LIN {X 0,Y 684.973,Z 1061.828,A -85,B 0,C 180,E1 30898.463,E2 30898.463} C_VEL
LIN {X 0,Y 683.766,Z 1083.483,A -85,B 0,C 180,E1 30896.498,E2 30896.498} C_VEL
LIN {X 0,Y 682.983,Z 1099.696,A -85,B 0,C 180,E1 30894.844,E2 30894.844} C_VEL
LIN {X 0,Y 682.192,Z 1116.492,A -85,B 0,C 180,E1 30892.946,E2 30892.946} C_VEL
LIN {X 0,Y 681.497,Z 1132.898,A -85,B 0,C 180,E1 30890.835,E2 30890.835} C_VEL
LIN {X 0,Y 681.037,Z 1145.572,A -85,B 0,C 180,E1 30889,E2 30889} C_VEL
LIN {X 0,Y 680.644,Z 1157.898,A -85,B 0,C 180,E1 30886.992,E2 30886.992} C_VEL
LIN {X 0,Y 680.337,Z 1169.84,A -85,B 0,C 180,E1 30884.729,E2 30884.729} C_VEL
LIN {X 0,Y 680.158,Z 1178.438,A -85,B 0,C 180,E1 30882.825,E2 30882.825} C_VEL
LIN {X 0,Y 680.019,Z 1186.223,A -85,B 0,C 180,E1 30880.819,E2 30880.819} C_VEL
LIN {X 0,Y 679.964,Z 1193.354,A -85,B 0,C 180,E1 30878.541,E2 30878.541} C_VEL
LIN {X 0,Y 679.926,Z 1198.83,A -85,B 0,C 180,E1 30876.216,E2 30876.216} C_VEL
LIN {X 0,Y 679.913,Z 1202.374,A -85,B 0,C 180,E1 30874.048,E2 30874.048} C_VEL
LIN {X 0,Y 679.907,Z 1204.494,A -85,B 0,C 180,E1 30871.77,E2 30871.77} C_VEL
LIN {X 0,Y 679.891,Z 1204.872,A -85,B 0,C 180,E1 30869.494,E2 30869.494} C_VEL
LIN {X 0,Y 679.907,Z 1203.956,A -85,B 0,C 180,E1 30867.471,E2 30867.471} C_VEL
LIN {X 0,Y 679.911,Z 1201.428,A -85,B 0,C 180,E1 30865.276,E2 30865.276} C_VEL
LIN {X 0,Y 679.934,Z 1197.152,A -85,B 0,C 180,E1 30862.989,E2 30862.989} C_VEL
LIN {X 0,Y 679.978,Z 1191.385,A -85,B 0,C 180,E1 30860.777,E2 30860.777} C_VEL
LIN {X 0,Y 680.067,Z 1184.278,A -85,B 0,C 180,E1 30858.638,E2 30858.638} C_VEL
LIN {X 0,Y 680.24,Z 1173.938,A -85,B 0,C 180,E1 30856.138,E2 30856.138} C_VEL
LIN {X 0,Y 680.464,Z 1164.538,A -85,B 0,C 180,E1 30854.227,E2 30854.227} C_VEL
LIN {X 0,Y 680.75,Z 1154.23,A -85,B 0,C 180,E1 30852.388,E2 30852.388} C_VEL
LIN {X 0,Y 681.149,Z 1141.939,A -85,B 0,C 180,E1 30850.447,E2 30850.447} C_VEL
LIN {X 0,Y 681.795,Z 1125.467,A -85,B 0,C 180,E1 30848.177,E2 30848.177} C_VEL
LIN {X 0,Y 682.441,Z 1111.072,A -85,B 0,C 180,E1 30846.423,E2 30846.423} C_VEL
LIN {X 0,Y 683.272,Z 1093.721,A -85,B 0,C 180,E1 30844.518,E2 30844.518} C_VEL
LIN {X 0,Y 684.268,Z 1074.724,A -85,B 0,C 180,E1 30842.679,E2 30842.679} C_VEL
LIN {X 0,Y 685.156,Z 1057.953,A -85,B 0,C 180,E1 30841.212,E2 30841.212} C_VEL
LIN {X 0,Y 686.26,Z 1038.594,A -85,B 0,C 180,E1 30839.679,E2 30839.679} C_VEL
LIN {X 0,Y 687.621,Z 1015.181,A -85,B 0,C 180,E1 30838.043,E2 30838.043} C_VEL
LIN {X 0,Y 688.735,Z 995.45,A -85,B 0,C 180,E1 30836.818,E2 30836.818} C_VEL
LIN {X 0,Y 689.843,Z 975.498,A -85,B 0,C 180,E1 30835.709,E2 30835.709} C_VEL
LIN {X 0,Y 691.118,Z 951.696,A -85,B 0,C 180,E1 30834.54,E2 30834.54} C_VEL
LIN {X 0,Y 692.334,Z 926.433,A -85,B 0,C 180,E1 30833.487,E2 30833.487} C_VEL
LIN {X 0,Y 693.317,Z 904.148,A -85,B 0,C 180,E1 30832.695,E2 30832.695} C_VEL
LIN {X 0,Y 694.253,Z 881.072,A -85,B 0,C 180,E1 30832.002,E2 30832.002} C_VEL
LIN {X 0,Y 695.165,Z 854.15,A -85,B 0,C 180,E1 30831.357,E2 30831.357} C_VEL
LIN {X 0,Y 695.824,Z 826.984,A -85,B 0,C 180,E1 30830.881,E2 30830.881} C_VEL
LIN {X 0,Y 698.219,Z 604.951,A -85,B 0,C 180,E1 30828.078,E2 30828.078} C_VEL
LIN {X 0,Y 700.483,Z 400.768,A -85,B 0,C 180,E1 30825.432,E2 30825.432} C_VEL
LIN {X 0,Y 700.65,Z 371.916,A -85,B 0,C 180,E1 30825.038,E2 30825.038} C_VEL
LIN {X 0,Y 697.923,Z 362.231,A -85,B 0,C 180,E1 30824.675,E2 30824.675} C_VEL
LIN {X 0,Y 690.097,Z 350.376,A -85,B 0,C 180,E1 30823.819,E2 30823.819} C_VEL
LIN {X 0,Y 683.625,Z 336.783,A -85,B 0,C 180,E1 30822.171,E2 30822.171} C_VEL
LIN {X 0,Y 681.952,Z 333.226,A -85,B 0,C 180,E1 30821.731,E2 30821.731} C_VEL
LIN {X 0,Y 680.493,Z 329.763,A -85,B 0,C 180,E1 30821.314,E2 30821.314} C_VEL
LIN {X 0,Y 680.459,Z 329.472,A -85,B 0,C 180,E1 30821.171,E2 30821.171} C_VEL
LIN {X 0,Y 680.503,Z 329.468,A -85,B 0,C 180,E1 30818.107,E2 30818.107} C_VEL
LIN {X 0,Y 680.45,Z 329.469,A -85,B 0,C 180,E1 30815.361,E2 30815.361} C_VEL
LIN {X 0,Y 680.488,Z 329.464,A -85,B 0,C 180,E1 30812.657,E2 30812.657} C_VEL
LIN {X 0,Y 680.469,Z 329.468,A -85,B 0,C 180,E1 30809.557,E2 30809.557} C_VEL
LIN {X 0,Y 680.449,Z 329.447,A -85,B 0,C 180,E1 30807.005,E2 30807.005} C_VEL
LIN {X 0,Y 680.526,Z 329.463,A -85,B 0,C 180,E1 30804.108,E2 30804.108} C_VEL
LIN {X 0,Y 680.462,Z 329.465,A -85,B 0,C 180,E1 30801.191,E2 30801.191} C_VEL
LIN {X 0,Y 680.459,Z 329.459,A -85,B 0,C 180,E1 30798.595,E2 30798.595} C_VEL
LIN {X 0,Y 680.526,Z 329.458,A -85,B 0,C 180,E1 30795.598,E2 30795.598} C_VEL
LIN {X 0,Y 680.454,Z 329.448,A -85,B 0,C 180,E1 30792.734,E2 30792.734} C_VEL
LIN {X 0,Y 680.494,Z 329.459,A -85,B 0,C 180,E1 30789.985,E2 30789.985} C_VEL
LIN {X 0,Y 680.474,Z 329.447,A -85,B 0,C 180,E1 30786.92,E2 30786.92} C_VEL
LIN {X 0,Y 680.458,Z 329.464,A -85,B 0,C 180,E1 30784.298,E2 30784.298} C_VEL
LIN {X 0,Y 680.527,Z 329.443,A -85,B 0,C 180,E1 30781.347,E2 30781.347} C_VEL
LIN {X 0,Y 680.461,Z 329.465,A -85,B 0,C 180,E1 30778.4,E2 30778.4} C_VEL
LIN {X 0,Y 680.49,Z 329.442,A -85,B 0,C 180,E1 30775.618,E2 30775.618} C_VEL
LIN {X 0,Y 680.477,Z 329.463,A -85,B 0,C 180,E1 30772.485,E2 30772.485} C_VEL
LIN {X 0,Y 680.465,Z 329.451,A -85,B 0,C 180,E1 30769.758,E2 30769.758} C_VEL
LIN {X 0,Y 680.527,Z 329.454,A -85,B 0,C 180,E1 30766.749,E2 30766.749} C_VEL
LIN {X 0,Y 680.462,Z 329.464,A -85,B 0,C 180,E1 30763.876,E2 30763.876} C_VEL
LIN {X 0,Y 680.512,Z 329.449,A -85,B 0,C 180,E1 30761.051,E2 30761.051} C_VEL
LIN {X 0,Y 680.475,Z 329.464,A -85,B 0,C 180,E1 30757.994,E2 30757.994} C_VEL
LIN {X 0,Y 680.474,Z 329.458,A -85,B 0,C 180,E1 30755.238,E2 30755.238} C_VEL
LIN {X 0,Y 680.512,Z 329.467,A -85,B 0,C 180,E1 30752.144,E2 30752.144} C_VEL
LIN {X 0,Y 680.466,Z 329.463,A -85,B 0,C 180,E1 30749.39,E2 30749.39} C_VEL
LIN {X 0,Y 679.48,Z 329.589,A -85,B 0,C 180,E1 30748.742,E2 30748.742} C_VEL
LIN {X 0,Y 673.099,Z 330.39,A -85,B 0,C 180,E1 30746.924,E2 30746.924} C_VEL
LIN {X 0,Y 672.588,Z 330.454,A -85,B 0,C 180,E1 30746.452,E2 30746.452} C_VEL
LIN {X 0,Y 672.558,Z 330.625,A -85,B 0,C 180,E1 30745.555,E2 30745.555} C_VEL
LIN {X 0,Y 673.93,Z 334.074,A -85,B 0,C 180,E1 30745.129,E2 30745.129} C_VEL
LIN {X 0,Y 677.255,Z 341.083,A -85,B 0,C 180,E1 30744.248,E2 30744.248} C_VEL
LIN {X 0,Y 689.877,Z 359.457,A -85,B 0,C 180,E1 30742.854,E2 30742.854} C_VEL
LIN {X 0,Y 695.097,Z 367.633,A -85,B 0,C 180,E1 30742.294,E2 30742.294} C_VEL
LIN {X 0,Y 692.503,Z 574.54,A -85,B 0,C 180,E1 30739.585,E2 30739.585} C_VEL
LIN {X 0,Y 689.933,Z 798.204,A -85,B 0,C 180,E1 30736.745,E2 30736.745} C_VEL
LIN {X 0,Y 689.322,Z 828.688,A -85,B 0,C 180,E1 30736.308,E2 30736.308} C_VEL
LIN {X 0,Y 688.525,Z 853.699,A -85,B 0,C 180,E1 30735.805,E2 30735.805} C_VEL
LIN {X 0,Y 687.518,Z 880.23,A -85,B 0,C 180,E1 30735.112,E2 30735.112} C_VEL
LIN {X 0,Y 686.268,Z 907.112,A -85,B 0,C 180,E1 30734.225,E2 30734.225} C_VEL
LIN {X 0,Y 685.119,Z 929.491,A -85,B 0,C 180,E1 30733.348,E2 30733.348} C_VEL
LIN {X 0,Y 683.72,Z 954.189,A -85,B 0,C 180,E1 30732.219,E2 30732.219} C_VEL
LIN {X 0,Y 682.144,Z 979.486,A -85,B 0,C 180,E1 30730.873,E2 30730.873} C_VEL
LIN {X 0,Y 680.693,Z 1002.914,A -85,B 0,C 180,E1 30729.436,E2 30729.436} C_VEL
LIN {X 0,Y 679.296,Z 1024.873,A -85,B 0,C 180,E1 30727.911,E2 30727.911} C_VEL
LIN {X 0,Y 677.913,Z 1046.47,A -85,B 0,C 180,E1 30726.215,E2 30726.215} C_VEL
LIN {X 0,Y 676.678,Z 1067.352,A -85,B 0,C 180,E1 30724.363,E2 30724.363} C_VEL
LIN {X 0,Y 675.512,Z 1086.947,A -85,B 0,C 180,E1 30722.399,E2 30722.399} C_VEL
LIN {X 0,Y 674.581,Z 1105,A -85,B 0,C 180,E1 30720.36,E2 30720.36} C_VEL
LIN {X 0,Y 673.743,Z 1122.087,A -85,B 0,C 180,E1 30718.159,E2 30718.159} C_VEL
LIN {X 0,Y 673.134,Z 1136.715,A -85,B 0,C 180,E1 30716.014,E2 30716.014} C_VEL
LIN {X 0,Y 672.647,Z 1150.472,A -85,B 0,C 180,E1 30713.696,E2 30713.696} C_VEL
LIN {X 0,Y 672.343,Z 1161.747,A -85,B 0,C 180,E1 30711.459,E2 30711.459} C_VEL
LIN {X 0,Y 672.134,Z 1170.61,A -85,B 0,C 180,E1 30709.41,E2 30709.41} C_VEL
LIN {X 0,Y 672.014,Z 1178.571,A -85,B 0,C 180,E1 30707.208,E2 30707.208} C_VEL
LIN {X 0,Y 671.96,Z 1185.341,A -85,B 0,C 180,E1 30704.829,E2 30704.829} C_VEL
LIN {X 0,Y 671.927,Z 1190.109,A -85,B 0,C 180,E1 30702.548,E2 30702.548} C_VEL
LIN {X 0,Y 671.919,Z 1193.274,A -85,B 0,C 180,E1 30700.286,E2 30700.286} C_VEL
LIN {X 0,Y 671.908,Z 1194.7,A -85,B 0,C 180,E1 30698.127,E2 30698.127} C_VEL
LIN {X 0,Y 671.913,Z 1194.819,A -85,B 0,C 180,E1 30696.236,E2 30696.236} C_VEL
LIN {X 0,Y 671.913,Z 1193.788,A -85,B 0,C 180,E1 30694.181,E2 30694.181} C_VEL
LIN {X 0,Y 671.92,Z 1190.996,A -85,B 0,C 180,E1 30691.876,E2 30691.876} C_VEL
LIN {X 0,Y 671.938,Z 1186.49,A -85,B 0,C 180,E1 30689.574,E2 30689.574} C_VEL
LIN {X 0,Y 671.998,Z 1180.619,A -85,B 0,C 180,E1 30687.356,E2 30687.356} C_VEL
LIN {X 0,Y 672.108,Z 1172.449,A -85,B 0,C 180,E1 30684.965,E2 30684.965} C_VEL
LIN {X 0,Y 672.308,Z 1163.087,A -85,B 0,C 180,E1 30682.738,E2 30682.738} C_VEL
LIN {X 0,Y 672.574,Z 1152.894,A -85,B 0,C 180,E1 30680.675,E2 30680.675} C_VEL
LIN {X 0,Y 672.996,Z 1140.618,A -85,B 0,C 180,E1 30678.517,E2 30678.517} C_VEL
LIN {X 0,Y 673.553,Z 1126.357,A -85,B 0,C 180,E1 30676.348,E2 30676.348} C_VEL
LIN {X 0,Y 674.262,Z 1110.628,A -85,B 0,C 180,E1 30674.245,E2 30674.245} C_VEL
LIN {X 0,Y 675.225,Z 1092.867,A -85,B 0,C 180,E1 30672.15,E2 30672.15} C_VEL
LIN {X 0,Y 676.3,Z 1073.164,A -85,B 0,C 180,E1 30670.104,E2 30670.104} C_VEL
LIN {X 0,Y 677.596,Z 1051.897,A -85,B 0,C 180,E1 30668.154,E2 30668.154} C_VEL
LIN {X 0,Y 678.995,Z 1029.504,A -85,B 0,C 180,E1 30666.343,E2 30666.343} C_VEL
LIN {X 0,Y 680.508,Z 1006.177,A -85,B 0,C 180,E1 30664.687,E2 30664.687} C_VEL
LIN {X 0,Y 682.022,Z 981.614,A -85,B 0,C 180,E1 30663.158,E2 30663.158} C_VEL
LIN {X 0,Y 683.636,Z 955.647,A -85,B 0,C 180,E1 30661.762,E2 30661.762} C_VEL
LIN {X 0,Y 685.083,Z 930.161,A -85,B 0,C 180,E1 30660.591,E2 30660.591} C_VEL
LIN {X 0,Y 686.276,Z 906.976,A -85,B 0,C 180,E1 30659.68,E2 30659.68} C_VEL
LIN {X 0,Y 687.523,Z 880.087,A -85,B 0,C 180,E1 30658.793,E2 30658.793} C_VEL
LIN {X 0,Y 688.539,Z 853.473,A -85,B 0,C 180,E1 30658.101,E2 30658.101} C_VEL
LIN {X 0,Y 689.323,Z 828.529,A -85,B 0,C 180,E1 30657.598,E2 30657.598} C_VEL
LIN {X 0,Y 689.945,Z 796.974,A -85,B 0,C 180,E1 30657.15,E2 30657.15} C_VEL
LIN {X 0,Y 692.503,Z 574.702,A -85,B 0,C 180,E1 30654.328,E2 30654.328} C_VEL
LIN {X 0,Y 695.099,Z 367.462,A -85,B 0,C 180,E1 30651.614,E2 30651.614} C_VEL
LIN {X 0,Y 684.64,Z 351.816,A -85,B 0,C 180,E1 30650.488,E2 30650.488} C_VEL
LIN {X 0,Y 677.093,Z 340.807,A -85,B 0,C 180,E1 30649.641,E2 30649.641} C_VEL
LIN {X 0,Y 673.916,Z 334.126,A -85,B 0,C 180,E1 30648.785,E2 30648.785} C_VEL
LIN {X 0,Y 672.529,Z 330.601,A -85,B 0,C 180,E1 30648.352,E2 30648.352} C_VEL
LIN {X 0,Y 672.5,Z 330.462,A -85,B 0,C 180,E1 30645.192,E2 30645.192} C_VEL
LIN {X 0,Y 672.483,Z 330.449,A -85,B 0,C 180,E1 30642.689,E2 30642.689} C_VEL
LIN {X 0,Y 672.525,Z 330.46,A -85,B 0,C 180,E1 30640.034,E2 30640.034} C_VEL
LIN {X 0,Y 672.507,Z 330.456,A -85,B 0,C 180,E1 30637.024,E2 30637.024} C_VEL
LIN {X 0,Y 672.486,Z 330.453,A -85,B 0,C 180,E1 30634.506,E2 30634.506} C_VEL
LIN {X 0,Y 672.522,Z 330.454,A -85,B 0,C 180,E1 30631.858,E2 30631.858} C_VEL
LIN {X 0,Y 672.507,Z 330.439,A -85,B 0,C 180,E1 30628.798,E2 30628.798} C_VEL
LIN {X 0,Y 672.49,Z 330.45,A -85,B 0,C 180,E1 30626.206,E2 30626.206} C_VEL
LIN {X 0,Y 672.56,Z 330.445,A -85,B 0,C 180,E1 30623.388,E2 30623.388} C_VEL
LIN {X 0,Y 672.5,Z 330.447,A -85,B 0,C 180,E1 30620.451,E2 30620.451} C_VEL
LIN {X 0,Y 672.493,Z 330.457,A -85,B 0,C 180,E1 30617.91,E2 30617.91} C_VEL
LIN {X 0,Y 672.587,Z 330.454,A -85,B 0,C 180,E1 30614.992,E2 30614.992} C_VEL
LIN {X 0,Y 672.495,Z 330.456,A -85,B 0,C 180,E1 30612.102,E2 30612.102} C_VEL
LIN {X 0,Y 672.499,Z 330.451,A -85,B 0,C 180,E1 30609.586,E2 30609.586} C_VEL
LIN {X 0,Y 672.576,Z 330.446,A -85,B 0,C 180,E1 30606.659,E2 30606.659} C_VEL
LIN {X 0,Y 672.496,Z 330.455,A -85,B 0,C 180,E1 30603.836,E2 30603.836} C_VEL
LIN {X 0,Y 672.507,Z 330.455,A -85,B 0,C 180,E1 30601.278,E2 30601.278} C_VEL
LIN {X 0,Y 672.544,Z 330.454,A -85,B 0,C 180,E1 30598.211,E2 30598.211} C_VEL
LIN {X 0,Y 672.495,Z 330.449,A -85,B 0,C 180,E1 30595.48,E2 30595.48} C_VEL
LIN {X 0,Y 672.532,Z 330.457,A -85,B 0,C 180,E1 30592.826,E2 30592.826} C_VEL
LIN {X 0,Y 672.516,Z 330.453,A -85,B 0,C 180,E1 30589.723,E2 30589.723} C_VEL
LIN {X 0,Y 672.497,Z 330.431,A -85,B 0,C 180,E1 30587.113,E2 30587.113} C_VEL
LIN {X 0,Y 672.589,Z 330.454,A -85,B 0,C 180,E1 30584.213,E2 30584.213} C_VEL
LIN {X 0,Y 672.501,Z 330.433,A -85,B 0,C 180,E1 30581.267,E2 30581.267} C_VEL
LIN {X 0,Y 672.509,Z 330.453,A -85,B 0,C 180,E1 30578.729,E2 30578.729} C_VEL
LIN {X 0,Y 672.572,Z 330.426,A -85,B 0,C 180,E1 30575.775,E2 30575.775} C_VEL
LIN {X 0,Y 672.503,Z 330.456,A -85,B 0,C 180,E1 30572.937,E2 30572.937} C_VEL
LIN {X 0,Y 672.518,Z 330.456,A -85,B 0,C 180,E1 30570.421,E2 30570.421} C_VEL
LIN {X 0,Y 672.54,Z 330.449,A -85,B 0,C 180,E1 30567.295,E2 30567.295} C_VEL
LIN {X 0,Y 672.505,Z 330.458,A -85,B 0,C 180,E1 30564.664,E2 30564.664} C_VEL
LIN {X 0,Y 672.554,Z 330.459,A -85,B 0,C 180,E1 30561.904,E2 30561.904} C_VEL
LIN {X 0,Y 672.607,Z 330.647,A -85,B 0,C 180,E1 30559.373,E2 30559.373} C_VEL
LIN {X 0,Y 673.724,Z 333.765,A -85,B 0,C 180,E1 30559.006,E2 30559.006} C_VEL
LIN {X 0,Y 674.752,Z 335.745,A -85,B 0,C 180,E1 30558.743,E2 30558.743} C_VEL
LIN {X 0,Y 680.467,Z 347.718,A -85,B 0,C 180,E1 30557.244,E2 30557.244} C_VEL
LIN {X 0,Y 682.245,Z 351.275,A -85,B 0,C 180,E1 30556.838,E2 30556.838} C_VEL
LIN {X 0,Y 693.378,Z 368.094,A -85,B 0,C 180,E1 30555.621,E2 30555.621} C_VEL
LIN {X 0,Y 695.107,Z 375.521,A -85,B 0,C 180,E1 30555.368,E2 30555.368} C_VEL
LIN {X 0,Y 692.461,Z 588.144,A -85,B 0,C 180,E1 30552.583,E2 30552.583} C_VEL
LIN {X 0,Y 689.897,Z 811.206,A -85,B 0,C 180,E1 30549.752,E2 30549.752} C_VEL
LIN {X 0,Y 689.263,Z 840.839,A -85,B 0,C 180,E1 30549.316,E2 30549.316} C_VEL
LIN {X 0,Y 688.458,Z 865.479,A -85,B 0,C 180,E1 30548.808,E2 30548.808} C_VEL
LIN {X 0,Y 687.469,Z 891.275,A -85,B 0,C 180,E1 30548.126,E2 30548.126} C_VEL
LIN {X 0,Y 686.224,Z 918.056,A -85,B 0,C 180,E1 30547.234,E2 30547.234} C_VEL
LIN {X 0,Y 685.095,Z 939.496,A -85,B 0,C 180,E1 30546.389,E2 30546.389} C_VEL
LIN {X 0,Y 683.955,Z 959.73,A -85,B 0,C 180,E1 30545.476,E2 30545.476} C_VEL
LIN {X 0,Y 682.725,Z 980.341,A -85,B 0,C 180,E1 30544.423,E2 30544.423} C_VEL
LIN {X 0,Y 681.198,Z 1004.941,A -85,B 0,C 180,E1 30542.994,E2 30542.994} C_VEL
LIN {X 0,Y 679.763,Z 1026.922,A -85,B 0,C 180,E1 30541.527,E2 30541.527} C_VEL
LIN {X 0,Y 678.597,Z 1045.714,A -85,B 0,C 180,E1 30540.125,E2 30540.125} C_VEL
LIN {X 0,Y 677.317,Z 1066.77,A -85,B 0,C 180,E1 30538.376,E2 30538.376} C_VEL
LIN {X 0,Y 676.137,Z 1085.458,A -85,B 0,C 180,E1 30536.62,E2 30536.62} C_VEL
LIN {X 0,Y 675.284,Z 1101.394,A -85,B 0,C 180,E1 30534.96,E2 30534.96} C_VEL
LIN {X 0,Y 674.297,Z 1120.139,A -85,B 0,C 180,E1 30532.769,E2 30532.769} C_VEL
LIN {X 0,Y 673.635,Z 1134.464,A -85,B 0,C 180,E1 30530.868,E2 30530.868} C_VEL
LIN {X 0,Y 673.123,Z 1147.17,A -85,B 0,C 180,E1 30528.984,E2 30528.984} C_VEL
LIN {X 0,Y 672.639,Z 1160.814,A -85,B 0,C 180,E1 30526.672,E2 30526.672} C_VEL
LIN {X 0,Y 672.363,Z 1171.073,A -85,B 0,C 180,E1 30524.643,E2 30524.643} C_VEL
LIN {X 0,Y 672.176,Z 1179.154,A -85,B 0,C 180,E1 30522.805,E2 30522.805} C_VEL
LIN {X 0,Y 672.029,Z 1186.719,A -85,B 0,C 180,E1 30520.805,E2 30520.805} C_VEL
LIN {X 0,Y 671.97,Z 1193.595,A -85,B 0,C 180,E1 30518.557,E2 30518.557} C_VEL
LIN {X 0,Y 671.928,Z 1198.936,A -85,B 0,C 180,E1 30516.236,E2 30516.236} C_VEL
LIN {X 0,Y 671.915,Z 1202.371,A -85,B 0,C 180,E1 30514.096,E2 30514.096} C_VEL
LIN {X 0,Y 671.907,Z 1204.494,A -85,B 0,C 180,E1 30511.791,E2 30511.791} C_VEL
LIN {X 0,Y 671.891,Z 1204.872,A -85,B 0,C 180,E1 30509.488,E2 30509.488} C_VEL
LIN {X 0,Y 671.907,Z 1203.953,A -85,B 0,C 180,E1 30507.441,E2 30507.441} C_VEL
LIN {X 0,Y 671.914,Z 1201.428,A -85,B 0,C 180,E1 30505.22,E2 30505.22} C_VEL
LIN {X 0,Y 671.941,Z 1197.152,A -85,B 0,C 180,E1 30502.906,E2 30502.906} C_VEL
LIN {X 0,Y 671.991,Z 1191.382,A -85,B 0,C 180,E1 30500.666,E2 30500.666} C_VEL
LIN {X 0,Y 672.091,Z 1184.278,A -85,B 0,C 180,E1 30498.501,E2 30498.501} C_VEL
LIN {X 0,Y 672.277,Z 1174.341,A -85,B 0,C 180,E1 30496.058,E2 30496.058} C_VEL
LIN {X 0,Y 672.534,Z 1164.539,A -85,B 0,C 180,E1 30494.036,E2 30494.036} C_VEL
LIN {X 0,Y 672.865,Z 1154.231,A -85,B 0,C 180,E1 30492.175,E2 30492.175} C_VEL
LIN {X 0,Y 673.319,Z 1141.941,A -85,B 0,C 180,E1 30490.21,E2 30490.21} C_VEL
LIN {X 0,Y 674.025,Z 1125.809,A -85,B 0,C 180,E1 30487.957,E2 30487.957} C_VEL
LIN {X 0,Y 674.751,Z 1111.074,A -85,B 0,C 180,E1 30486.138,E2 30486.138} C_VEL
LIN {X 0,Y 675.713,Z 1093.722,A -85,B 0,C 180,E1 30484.213,E2 30484.213} C_VEL
LIN {X 0,Y 676.817,Z 1074.328,A -85,B 0,C 180,E1 30482.315,E2 30482.315} C_VEL
LIN {X 0,Y 677.816,Z 1057.658,A -85,B 0,C 180,E1 30480.845,E2 30480.845} C_VEL
LIN {X 0,Y 679.089,Z 1037.983,A -85,B 0,C 180,E1 30479.276,E2 30479.276} C_VEL
LIN {X 0,Y 680.588,Z 1014.456,A -85,B 0,C 180,E1 30477.623,E2 30477.623} C_VEL
LIN {X 0,Y 681.824,Z 994.65,A -85,B 0,C 180,E1 30476.387,E2 30476.387} C_VEL
LIN {X 0,Y 683.13,Z 973.171,A -85,B 0,C 180,E1 30475.193,E2 30475.193} C_VEL
LIN {X 0,Y 684.731,Z 946.23,A -85,B 0,C 180,E1 30473.9,E2 30473.9} C_VEL
LIN {X 0,Y 685.855,Z 925.015,A -85,B 0,C 180,E1 30473.027,E2 30473.027} C_VEL
LIN {X 0,Y 686.852,Z 904.075,A -85,B 0,C 180,E1 30472.28,E2 30472.28} C_VEL
LIN {X 0,Y 687.876,Z 880.996,A -85,B 0,C 180,E1 30471.584,E2 30471.584} C_VEL
LIN {X 0,Y 688.887,Z 854.068,A -85,B 0,C 180,E1 30470.936,E2 30470.936} C_VEL
LIN {X 0,Y 689.603,Z 827.166,A -85,B 0,C 180,E1 30470.463,E2 30470.463} C_VEL
LIN {X 0,Y 692.23,Z 607.496,A -85,B 0,C 180,E1 30467.666,E2 30467.666} C_VEL
LIN {X 0,Y 694.741,Z 403.536,A -85,B 0,C 180,E1 30465.004,E2 30465.004} C_VEL
LIN {X 0,Y 694.947,Z 374.179,A -85,B 0,C 180,E1 30464.599,E2 30464.599} C_VEL
LIN {X 0,Y 692.936,Z 367.15,A -85,B 0,C 180,E1 30464.328,E2 30464.328} C_VEL
LIN {X 0,Y 681.806,Z 350.663,A -85,B 0,C 180,E1 30463.111,E2 30463.111} C_VEL
LIN {X 0,Y 676.085,Z 338.5,A -85,B 0,C 180,E1 30461.609,E2 30461.609} C_VEL
LIN {X 0,Y 673.718,Z 333.754,A -85,B 0,C 180,E1 30460.995,E2 30460.995} C_VEL
LIN {X 0,Y 672.585,Z 330.454,A -85,B 0,C 180,E1 30460.598,E2 30460.598} C_VEL
LIN {X 0,Y 672.518,Z 330.46,A -85,B 0,C 180,E1 30457.667,E2 30457.667} C_VEL
LIN {X 0,Y 672.521,Z 330.457,A -85,B 0,C 180,E1 30455.023,E2 30455.023} C_VEL
LIN {X 0,Y 672.567,Z 330.436,A -85,B 0,C 180,E1 30451.955,E2 30451.955} C_VEL
LIN {X 0,Y 672.513,Z 330.456,A -85,B 0,C 180,E1 30449.188,E2 30449.188} C_VEL
LIN {X 0,Y 672.548,Z 330.433,A -85,B 0,C 180,E1 30446.489,E2 30446.489} C_VEL
LIN {X 0,Y 672.532,Z 330.441,A -85,B 0,C 180,E1 30443.389,E2 30443.389} C_VEL
LIN {X 0,Y 672.517,Z 330.452,A -85,B 0,C 180,E1 30440.723,E2 30440.723} C_VEL
LIN {X 0,Y 672.586,Z 330.432,A -85,B 0,C 180,E1 30437.744,E2 30437.744} C_VEL
LIN {X 0,Y 672.516,Z 330.455,A -85,B 0,C 180,E1 30434.817,E2 30434.817} C_VEL
LIN {X 0,Y 672.546,Z 330.431,A -85,B 0,C 180,E1 30432.101,E2 30432.101} C_VEL
LIN {X 0,Y 672.536,Z 330.453,A -85,B 0,C 180,E1 30428.981,E2 30428.981} C_VEL
LIN {X 0,Y 672.518,Z 330.436,A -85,B 0,C 180,E1 30426.317,E2 30426.317} C_VEL
LIN {X 0,Y 672.588,Z 330.451,A -85,B 0,C 180,E1 30423.324,E2 30423.324} C_VEL
LIN {X 0,Y 672.519,Z 330.446,A -85,B 0,C 180,E1 30420.426,E2 30420.426} C_VEL
LIN {X 0,Y 672.55,Z 330.451,A -85,B 0,C 180,E1 30417.699,E2 30417.699} C_VEL
LIN {X 0,Y 672.537,Z 330.449,A -85,B 0,C 180,E1 30414.54,E2 30414.54} C_VEL
LIN {X 0,Y 672.523,Z 330.448,A -85,B 0,C 180,E1 30411.88,E2 30411.88} C_VEL
LIN {X 0,Y 672.586,Z 330.443,A -85,B 0,C 180,E1 30408.856,E2 30408.856} C_VEL
LIN {X 0,Y 672.52,Z 330.437,A -85,B 0,C 180,E1 30405.975,E2 30405.975} C_VEL
LIN {X 0,Y 672.569,Z 330.448,A -85,B 0,C 180,E1 30403.148,E2 30403.148} C_VEL
LIN {X 0,Y 672.538,Z 330.441,A -85,B 0,C 180,E1 30400.095,E2 30400.095} C_VEL
LIN {X 0,Y 672.534,Z 330.449,A -85,B 0,C 180,E1 30397.352,E2 30397.352} C_VEL
LIN {X 0,Y 672.579,Z 330.456,A -85,B 0,C 180,E1 30394.272,E2 30394.272} C_VEL
LIN {X 0,Y 672.527,Z 330.456,A -85,B 0,C 180,E1 30391.397,E2 30391.397} C_VEL
LIN {X 0,Y 672.59,Z 330.451,A -85,B 0,C 180,E1 30388.446,E2 30388.446} C_VEL
LIN {X 0,Y 672.588,Z 330.454,A -85,B 0,C 180,E1 30386.452,E2 30386.452} C_VEL
LIN {X 0,Y 672.102,Z 331.387,A -85,B 0,C 180,E1 30386.073,E2 30386.073} C_VEL
LIN {X 0,Y 670.713,Z 334.55,A -85,B 0,C 180,E1 30385.627,E2 30385.627} C_VEL
LIN {X 0,Y 669.676,Z 339.366,A -85,B 0,C 180,E1 30385.186,E2 30385.186} C_VEL
LIN {X 0,Y 670.426,Z 343.195,A -85,B 0,C 180,E1 30384.864,E2 30384.864} C_VEL
LIN {X 0,Y 671.062,Z 344.162,A -85,B 0,C 180,E1 30384.777,E2 30384.777} C_VEL
LIN {X 0,Y 685.324,Z 364.863,A -85,B 0,C 180,E1 30383.168,E2 30383.168} C_VEL
LIN {X 0,Y 689.411,Z 371.316,A -85,B 0,C 180,E1 30382.72,E2 30382.72} C_VEL
LIN {X 0,Y 686.577,Z 577.085,A -85,B 0,C 180,E1 30380.006,E2 30380.006} C_VEL
LIN {X 0,Y 683.746,Z 801.158,A -85,B 0,C 180,E1 30377.138,E2 30377.138} C_VEL
LIN {X 0,Y 683.081,Z 829.724,A -85,B 0,C 180,E1 30376.718,E2 30376.718} C_VEL
LIN {X 0,Y 682.233,Z 854.24,A -85,B 0,C 180,E1 30376.218,E2 30376.218} C_VEL
LIN {X 0,Y 681.117,Z 880.908,A -85,B 0,C 180,E1 30375.515,E2 30375.515} C_VEL
LIN {X 0,Y 679.766,Z 907.246,A -85,B 0,C 180,E1 30374.637,E2 30374.637} C_VEL
LIN {X 0,Y 678.468,Z 930.362,A -85,B 0,C 180,E1 30373.722,E2 30373.722} C_VEL
LIN {X 0,Y 676.932,Z 955.274,A -85,B 0,C 180,E1 30372.57,E2 30372.57} C_VEL
LIN {X 0,Y 675.158,Z 981.101,A -85,B 0,C 180,E1 30371.174,E2 30371.174} C_VEL
LIN {X 0,Y 673.449,Z 1006.304,A -85,B 0,C 180,E1 30369.594,E2 30369.594} C_VEL
LIN {X 0,Y 671.747,Z 1030.189,A -85,B 0,C 180,E1 30367.878,E2 30367.878} C_VEL
LIN {X 0,Y 670.183,Z 1053.038,A -85,B 0,C 180,E1 30366.002,E2 30366.002} C_VEL
LIN {X 0,Y 668.781,Z 1073.707,A -85,B 0,C 180,E1 30364.077,E2 30364.077} C_VEL
LIN {X 0,Y 667.585,Z 1093.245,A -85,B 0,C 180,E1 30362.018,E2 30362.018} C_VEL
LIN {X 0,Y 666.538,Z 1111.192,A -85,B 0,C 180,E1 30359.869,E2 30359.869} C_VEL
LIN {X 0,Y 665.728,Z 1127.509,A -85,B 0,C 180,E1 30357.651,E2 30357.651} C_VEL
LIN {X 0,Y 665.073,Z 1142.106,A -85,B 0,C 180,E1 30355.369,E2 30355.369} C_VEL
LIN {X 0,Y 664.624,Z 1154.539,A -85,B 0,C 180,E1 30353.119,E2 30353.119} C_VEL
LIN {X 0,Y 664.315,Z 1165.1,A -85,B 0,C 180,E1 30350.898,E2 30350.898} C_VEL
LIN {X 0,Y 664.1,Z 1174.872,A -85,B 0,C 180,E1 30348.432,E2 30348.432} C_VEL
LIN {X 0,Y 663.991,Z 1182.019,A -85,B 0,C 180,E1 30346.175,E2 30346.175} C_VEL
LIN {X 0,Y 663.936,Z 1187.575,A -85,B 0,C 180,E1 30343.943,E2 30343.943} C_VEL
LIN {X 0,Y 663.911,Z 1191.776,A -85,B 0,C 180,E1 30341.554,E2 30341.554} C_VEL
LIN {X 0,Y 663.911,Z 1194.093,A -85,B 0,C 180,E1 30339.361,E2 30339.361} C_VEL
LIN {X 0,Y 663.917,Z 1194.997,A -85,B 0,C 180,E1 30336.92,E2 30336.92} C_VEL
LIN {X 0,Y 663.908,Z 1194.115,A -85,B 0,C 180,E1 30334.578,E2 30334.578} C_VEL
LIN {X 0,Y 663.917,Z 1191.741,A -85,B 0,C 180,E1 30332.33,E2 30332.33} C_VEL
LIN {X 0,Y 663.945,Z 1187.649,A -85,B 0,C 180,E1 30330,E2 30330} C_VEL
LIN {X 0,Y 663.995,Z 1182.079,A -85,B 0,C 180,E1 30327.756,E2 30327.756} C_VEL
LIN {X 0,Y 664.107,Z 1174.986,A -85,B 0,C 180,E1 30325.51,E2 30325.51} C_VEL
LIN {X 0,Y 664.287,Z 1165.422,A -85,B 0,C 180,E1 30323.084,E2 30323.084} C_VEL
LIN {X 0,Y 664.601,Z 1154.712,A -85,B 0,C 180,E1 30320.824,E2 30320.824} C_VEL
LIN {X 0,Y 665.038,Z 1142.686,A -85,B 0,C 180,E1 30318.641,E2 30318.641} C_VEL
LIN {X 0,Y 665.672,Z 1128.195,A -85,B 0,C 180,E1 30316.36,E2 30316.36} C_VEL
LIN {X 0,Y 666.434,Z 1112.763,A -85,B 0,C 180,E1 30314.243,E2 30314.243} C_VEL
LIN {X 0,Y 667.366,Z 1096.776,A -85,B 0,C 180,E1 30312.294,E2 30312.294} C_VEL
LIN {X 0,Y 668.507,Z 1077.805,A -85,B 0,C 180,E1 30310.244,E2 30310.244} C_VEL
LIN {X 0,Y 669.862,Z 1057.674,A -85,B 0,C 180,E1 30308.32,E2 30308.32} C_VEL
LIN {X 0,Y 671.35,Z 1035.847,A -85,B 0,C 180,E1 30306.476,E2 30306.476} C_VEL
LIN {X 0,Y 672.922,Z 1013.54,A -85,B 0,C 180,E1 30304.812,E2 30304.812} C_VEL
LIN {X 0,Y 674.585,Z 989.97,A -85,B 0,C 180,E1 30303.267,E2 30303.267} C_VEL
LIN {X 0,Y 676.279,Z 964.454,A -85,B 0,C 180,E1 30301.812,E2 30301.812} C_VEL
LIN {X 0,Y 678.056,Z 937.418,A -85,B 0,C 180,E1 30300.494,E2 30300.494} C_VEL
LIN {X 0,Y 679.539,Z 911.897,A -85,B 0,C 180,E1 30299.445,E2 30299.445} C_VEL
LIN {X 0,Y 680.699,Z 888.865,A -85,B 0,C 180,E1 30298.645,E2 30298.645} C_VEL
LIN {X 0,Y 681.857,Z 864.341,A -85,B 0,C 180,E1 30297.939,E2 30297.939} C_VEL
LIN {X 0,Y 682.868,Z 836.476,A -85,B 0,C 180,E1 30297.315,E2 30297.315} C_VEL
LIN {X 0,Y 683.558,Z 811.403,A -85,B 0,C 180,E1 30296.907,E2 30296.907} C_VEL
LIN {X 0,Y 686.384,Z 591.838,A -85,B 0,C 180,E1 30294.096,E2 30294.096} C_VEL
LIN {X 0,Y 689.268,Z 380.651,A -85,B 0,C 180,E1 30291.314,E2 30291.314} C_VEL
LIN {X 0,Y 689.262,Z 370.846,A -85,B 0,C 180,E1 30291.17,E2 30291.17} C_VEL
LIN {X 0,Y 676.384,Z 351.872,A -85,B 0,C 180,E1 30289.748,E2 30289.748} C_VEL
LIN {X 0,Y 668.701,Z 340.727,A -85,B 0,C 180,E1 30288.84,E2 30288.84} C_VEL
LIN {X 0,Y 665.738,Z 334.643,A -85,B 0,C 180,E1 30288.027,E2 30288.027} C_VEL
LIN {X 0,Y 664.608,Z 331.447,A -85,B 0,C 180,E1 30287.621,E2 30287.621} C_VEL
LIN {X 0,Y 664.545,Z 331.452,A -85,B 0,C 180,E1 30284.875,E2 30284.875} C_VEL
LIN {X 0,Y 664.564,Z 331.43,A -85,B 0,C 180,E1 30282.264,E2 30282.264} C_VEL
LIN {X 0,Y 664.568,Z 331.447,A -85,B 0,C 180,E1 30279.074,E2 30279.074} C_VEL
LIN {X 0,Y 664.547,Z 331.446,A -85,B 0,C 180,E1 30276.54,E2 30276.54} C_VEL
LIN {X 0,Y 664.594,Z 331.443,A -85,B 0,C 180,E1 30273.826,E2 30273.826} C_VEL
LIN {X 0,Y 664.562,Z 331.447,A -85,B 0,C 180,E1 30270.768,E2 30270.768} C_VEL
LIN {X 0,Y 664.547,Z 331.426,A -85,B 0,C 180,E1 30268.292,E2 30268.292} C_VEL
LIN {X 0,Y 664.613,Z 331.44,A -85,B 0,C 180,E1 30265.485,E2 30265.485} C_VEL
LIN {X 0,Y 664.558,Z 331.424,A -85,B 0,C 180,E1 30262.468,E2 30262.468} C_VEL
LIN {X 0,Y 664.553,Z 331.436,A -85,B 0,C 180,E1 30259.971,E2 30259.971} C_VEL
LIN {X 0,Y 664.642,Z 331.436,A -85,B 0,C 180,E1 30257.059,E2 30257.059} C_VEL
LIN {X 0,Y 664.558,Z 331.443,A -85,B 0,C 180,E1 30254.197,E2 30254.197} C_VEL
LIN {X 0,Y 664.556,Z 331.445,A -85,B 0,C 180,E1 30251.72,E2 30251.72} C_VEL
LIN {X 0,Y 664.64,Z 331.442,A -85,B 0,C 180,E1 30248.74,E2 30248.74} C_VEL
LIN {X 0,Y 664.555,Z 331.439,A -85,B 0,C 180,E1 30245.872,E2 30245.872} C_VEL
LIN {X 0,Y 664.572,Z 331.445,A -85,B 0,C 180,E1 30243.278,E2 30243.278} C_VEL
LIN {X 0,Y 664.582,Z 331.441,A -85,B 0,C 180,E1 30240.086,E2 30240.086} C_VEL
LIN {X 0,Y 664.558,Z 331.445,A -85,B 0,C 180,E1 30237.456,E2 30237.456} C_VEL
LIN {X 0,Y 664.637,Z 331.439,A -85,B 0,C 180,E1 30234.561,E2 30234.561} C_VEL
LIN {X 0,Y 664.565,Z 331.441,A -85,B 0,C 180,E1 30231.608,E2 30231.608} C_VEL
LIN {X 0,Y 664.564,Z 331.443,A -85,B 0,C 180,E1 30229.072,E2 30229.072} C_VEL
LIN {X 0,Y 664.634,Z 331.42,A -85,B 0,C 180,E1 30226.072,E2 30226.072} C_VEL
LIN {X 0,Y 664.564,Z 331.444,A -85,B 0,C 180,E1 30223.299,E2 30223.299} C_VEL
LIN {X 0,Y 664.576,Z 331.418,A -85,B 0,C 180,E1 30220.67,E2 30220.67} C_VEL
LIN {X 0,Y 664.589,Z 331.441,A -85,B 0,C 180,E1 30217.48,E2 30217.48} C_VEL
LIN {X 0,Y 664.561,Z 331.419,A -85,B 0,C 180,E1 30214.894,E2 30214.894} C_VEL
LIN {X 0,Y 664.622,Z 331.444,A -85,B 0,C 180,E1 30212.103,E2 30212.103} C_VEL
LIN {X 0,Y 664.574,Z 331.44,A -85,B 0,C 180,E1 30209.044,E2 30209.044} C_VEL
LIN {X 0,Y 664.572,Z 331.441,A -85,B 0,C 180,E1 30206.46,E2 30206.46} C_VEL
LIN {X 0,Y 664.635,Z 331.443,A -85,B 0,C 180,E1 30203.434,E2 30203.434} C_VEL
LIN {X 0,Y 664.567,Z 331.455,A -85,B 0,C 180,E1 30200.585,E2 30200.585} C_VEL
LIN {X 0,Y 664.617,Z 331.669,A -85,B 0,C 180,E1 30200.085,E2 30200.085} C_VEL
LIN {X 0,Y 665.94,Z 334.921,A -85,B 0,C 180,E1 30199.674,E2 30199.674} C_VEL
LIN {X 0,Y 666.942,Z 336.883,A -85,B 0,C 180,E1 30199.408,E2 30199.408} C_VEL
LIN {X 0,Y 673.766,Z 351.133,A -85,B 0,C 180,E1 30197.614,E2 30197.614} C_VEL
LIN {X 0,Y 686.84,Z 370.211,A -85,B 0,C 180,E1 30196.15,E2 30196.15} C_VEL
LIN {X 0,Y 688.472,Z 373.235,A -85,B 0,C 180,E1 30195.964,E2 30195.964} C_VEL
LIN {X 0,Y 689.447,Z 377.809,A -85,B 0,C 180,E1 30195.813,E2 30195.813} C_VEL
LIN {X 0,Y 686.547,Z 589.459,A -85,B 0,C 180,E1 30193.02,E2 30193.02} C_VEL
LIN {X 0,Y 683.729,Z 812.351,A -85,B 0,C 180,E1 30190.168,E2 30190.168} C_VEL
LIN {X 0,Y 683.036,Z 841.301,A -85,B 0,C 180,E1 30189.735,E2 30189.735} C_VEL
LIN {X 0,Y 682.182,Z 865.459,A -85,B 0,C 180,E1 30189.234,E2 30189.234} C_VEL
LIN {X 0,Y 681.099,Z 891.07,A -85,B 0,C 180,E1 30188.554,E2 30188.554} C_VEL
LIN {X 0,Y 679.737,Z 917.912,A -85,B 0,C 180,E1 30187.657,E2 30187.657} C_VEL
LIN {X 0,Y 678.49,Z 939.492,A -85,B 0,C 180,E1 30186.801,E2 30186.801} C_VEL
LIN {X 0,Y 677.241,Z 959.727,A -85,B 0,C 180,E1 30185.882,E2 30185.882} C_VEL
LIN {X 0,Y 675.886,Z 980.554,A -85,B 0,C 180,E1 30184.809,E2 30184.809} C_VEL
LIN {X 0,Y 674.235,Z 1004.939,A -85,B 0,C 180,E1 30183.379,E2 30183.379} C_VEL
LIN {X 0,Y 672.656,Z 1026.639,A -85,B 0,C 180,E1 30181.92,E2 30181.92} C_VEL
LIN {X 0,Y 671.37,Z 1045.271,A -85,B 0,C 180,E1 30180.52,E2 30180.52} C_VEL
LIN {X 0,Y 669.98,Z 1066.205,A -85,B 0,C 180,E1 30178.77,E2 30178.77} C_VEL
LIN {X 0,Y 668.655,Z 1085.189,A -85,B 0,C 180,E1 30176.969,E2 30176.969} C_VEL
LIN {X 0,Y 667.705,Z 1100.547,A -85,B 0,C 180,E1 30175.358,E2 30175.358} C_VEL
LIN {X 0,Y 666.721,Z 1118.009,A -85,B 0,C 180,E1 30173.323,E2 30173.323} C_VEL
LIN {X 0,Y 665.878,Z 1133.821,A -85,B 0,C 180,E1 30171.215,E2 30171.215} C_VEL
LIN {X 0,Y 665.317,Z 1146.017,A -85,B 0,C 180,E1 30169.398,E2 30169.398} C_VEL
LIN {X 0,Y 664.82,Z 1158.891,A -85,B 0,C 180,E1 30167.234,E2 30167.234} C_VEL
LIN {X 0,Y 664.423,Z 1170.664,A -85,B 0,C 180,E1 30164.912,E2 30164.912} C_VEL
LIN {X 0,Y 664.224,Z 1178.798,A -85,B 0,C 180,E1 30163.05,E2 30163.05} C_VEL
LIN {X 0,Y 664.054,Z 1186.419,A -85,B 0,C 180,E1 30161.024,E2 30161.024} C_VEL
LIN {X 0,Y 663.977,Z 1193.595,A -85,B 0,C 180,E1 30158.661,E2 30158.661} C_VEL
LIN {X 0,Y 663.932,Z 1198.968,A -85,B 0,C 180,E1 30156.293,E2 30156.293} C_VEL
LIN {X 0,Y 663.915,Z 1202.482,A -85,B 0,C 180,E1 30154.059,E2 30154.059} C_VEL
LIN {X 0,Y 663.907,Z 1204.549,A -85,B 0,C 180,E1 30151.726,E2 30151.726} C_VEL
LIN {X 0,Y 663.891,Z 1204.872,A -85,B 0,C 180,E1 30149.482,E2 30149.482} C_VEL
LIN {X 0,Y 663.908,Z 1203.95,A -85,B 0,C 180,E1 30147.41,E2 30147.41} C_VEL
LIN {X 0,Y 663.917,Z 1201.428,A -85,B 0,C 180,E1 30145.162,E2 30145.162} C_VEL
LIN {X 0,Y 663.948,Z 1197.152,A -85,B 0,C 180,E1 30142.82,E2 30142.82} C_VEL
LIN {X 0,Y 664.001,Z 1191.28,A -85,B 0,C 180,E1 30140.519,E2 30140.519} C_VEL
LIN {X 0,Y 664.109,Z 1183.959,A -85,B 0,C 180,E1 30138.273,E2 30138.273} C_VEL
LIN {X 0,Y 664.345,Z 1173.758,A -85,B 0,C 180,E1 30135.76,E2 30135.76} C_VEL
LIN {X 0,Y 664.618,Z 1164.076,A -85,B 0,C 180,E1 30133.751,E2 30133.751} C_VEL
LIN {X 0,Y 665.008,Z 1153.637,A -85,B 0,C 180,E1 30131.854,E2 30131.854} C_VEL
LIN {X 0,Y 665.631,Z 1139.567,A -85,B 0,C 180,E1 30129.605,E2 30129.605} C_VEL
LIN {X 0,Y 666.363,Z 1124.404,A -85,B 0,C 180,E1 30127.504,E2 30127.504} C_VEL
LIN {X 0,Y 667.166,Z 1109.516,A -85,B 0,C 180,E1 30125.661,E2 30125.661} C_VEL
LIN {X 0,Y 668.348,Z 1090.654,A -85,B 0,C 180,E1 30123.582,E2 30123.582} C_VEL
LIN {X 0,Y 669.435,Z 1073.313,A -85,B 0,C 180,E1 30121.886,E2 30121.886} C_VEL
LIN {X 0,Y 670.617,Z 1056.207,A -85,B 0,C 180,E1 30120.373,E2 30120.373} C_VEL
LIN {X 0,Y 672.188,Z 1034.208,A -85,B 0,C 180,E1 30118.627,E2 30118.627} C_VEL
LIN {X 0,Y 673.617,Z 1013.162,A -85,B 0,C 180,E1 30117.156,E2 30117.156} C_VEL
LIN {X 0,Y 674.999,Z 993.054,A -85,B 0,C 180,E1 30115.9,E2 30115.9} C_VEL
LIN {X 0,Y 676.708,Z 968.661,A -85,B 0,C 180,E1 30114.554,E2 30114.554} C_VEL
LIN {X 0,Y 678.238,Z 943.998,A -85,B 0,C 180,E1 30113.394,E2 30113.394} C_VEL
LIN {X 0,Y 679.403,Z 923.896,A -85,B 0,C 180,E1 30112.57,E2 30112.57} C_VEL
LIN {X 0,Y 680.471,Z 903.03,A -85,B 0,C 180,E1 30111.826,E2 30111.826} C_VEL
LIN {X 0,Y 681.603,Z 879.634,A -85,B 0,C 180,E1 30111.123,E2 30111.123} C_VEL
LIN {X 0,Y 682.719,Z 851.801,A -85,B 0,C 180,E1 30110.464,E2 30110.464} C_VEL
LIN {X 0,Y 683.44,Z 826.276,A -85,B 0,C 180,E1 30110.022,E2 30110.022} C_VEL
LIN {X 0,Y 686.307,Z 607.878,A -85,B 0,C 180,E1 30107.219,E2 30107.219} C_VEL
LIN {X 0,Y 689.069,Z 404.052,A -85,B 0,C 180,E1 30104.538,E2 30104.538} C_VEL
LIN {X 0,Y 689.288,Z 376.404,A -85,B 0,C 180,E1 30104.152,E2 30104.152} C_VEL
LIN {X 0,Y 687.98,Z 372.016,A -85,B 0,C 180,E1 30103.976,E2 30103.976} C_VEL
LIN {X 0,Y 677.362,Z 356.311,A -85,B 0,C 180,E1 30102.797,E2 30102.797} C_VEL
LIN {X 0,Y 673.316,Z 350.335,A -85,B 0,C 180,E1 30102.31,E2 30102.31} C_VEL
LIN {X 0,Y 666.327,Z 335.428,A -85,B 0,C 180,E1 30100.411,E2 30100.411} C_VEL
LIN {X 0,Y 664.707,Z 332.1,A -85,B 0,C 180,E1 30099.965,E2 30099.965} C_VEL
LIN {X 0,Y 664.589,Z 331.452,A -85,B 0,C 180,E1 30099.861,E2 30099.861} C_VEL
LIN {X 0,Y 664.576,Z 331.447,A -85,B 0,C 180,E1 30097.217,E2 30097.217} C_VEL
LIN {X 0,Y 664.651,Z 331.437,A -85,B 0,C 180,E1 30094.239,E2 30094.239} C_VEL
LIN {X 0,Y 664.573,Z 331.424,A -85,B 0,C 180,E1 30091.289,E2 30091.289} C_VEL
LIN {X 0,Y 664.606,Z 331.442,A -85,B 0,C 180,E1 30088.583,E2 30088.583} C_VEL
LIN {X 0,Y 664.591,Z 331.446,A -85,B 0,C 180,E1 30085.391,E2 30085.391} C_VEL
LIN {X 0,Y 664.579,Z 331.425,A -85,B 0,C 180,E1 30082.742,E2 30082.742} C_VEL
LIN {X 0,Y 664.644,Z 331.442,A -85,B 0,C 180,E1 30079.693,E2 30079.693} C_VEL
LIN {X 0,Y 664.576,Z 331.431,A -85,B 0,C 180,E1 30076.791,E2 30076.791} C_VEL
LIN {X 0,Y 664.64,Z 331.44,A -85,B 0,C 180,E1 30073.928,E2 30073.928} C_VEL
LIN {X 0,Y 664.584,Z 331.442,A -85,B 0,C 180,E1 30070.84,E2 30070.84} C_VEL
LIN {X 0,Y 664.595,Z 331.437,A -85,B 0,C 180,E1 30068.13,E2 30068.13} C_VEL
LIN {X 0,Y 664.604,Z 331.444,A -85,B 0,C 180,E1 30064.92,E2 30064.92} C_VEL
LIN {X 0,Y 664.583,Z 331.431,A -85,B 0,C 180,E1 30062.156,E2 30062.156} C_VEL
LIN {X 0,Y 664.648,Z 331.436,A -85,B 0,C 180,E1 30059.138,E2 30059.138} C_VEL
LIN {X 0,Y 664.578,Z 331.421,A -85,B 0,C 180,E1 30056.204,E2 30056.204} C_VEL
LIN {X 0,Y 664.65,Z 331.437,A -85,B 0,C 180,E1 30053.261,E2 30053.261} C_VEL
LIN {X 0,Y 664.586,Z 331.424,A -85,B 0,C 180,E1 30050.209,E2 30050.209} C_VEL
LIN {X 0,Y 664.614,Z 331.44,A -85,B 0,C 180,E1 30047.4,E2 30047.4} C_VEL
LIN {X 0,Y 664.606,Z 331.433,A -85,B 0,C 180,E1 30044.288,E2 30044.288} C_VEL
LIN {X 0,Y 664.588,Z 331.433,A -85,B 0,C 180,E1 30041.582,E2 30041.582} C_VEL
LIN {X 0,Y 664.65,Z 331.44,A -85,B 0,C 180,E1 30038.557,E2 30038.557} C_VEL
LIN {X 0,Y 664.585,Z 331.431,A -85,B 0,C 180,E1 30035.654,E2 30035.654} C_VEL
LIN {X 0,Y 664.642,Z 331.435,A -85,B 0,C 180,E1 30032.757,E2 30032.757} C_VEL
LIN {X 0,Y 664.598,Z 331.439,A -85,B 0,C 180,E1 30029.718,E2 30029.718} C_VEL
LIN {X 0,Y 664.61,Z 331.446,A -85,B 0,C 180,E1 30026.898,E2 30026.898} C_VEL
LIN {X 0,Y 664.675,Z 331.62,A -85,B 0,C 180,E1 30026.256,E2 30026.256} C_VEL
LIN {X 0,Y 666.126,Z 335.219,A -85,B 0,C 180,E1 30025.797,E2 30025.797} C_VEL
LIN {X 0,Y 669.098,Z 341.367,A -85,B 0,C 180,E1 30025.007,E2 30025.007} C_VEL
LIN {X 0,Y 671.062,Z 344.162,A -85,B 0,C 180,E1 30024.777,E2 30024.777} C_VEL
LIN {X 0,Y 673.813,Z 348.797,A -85,B 0,C 180,E1 30024.447,E2 30024.447} C_VEL
LIN {X 0,Y 676.672,Z 357.266,A -85,B 0,C 180,E1 30024.053,E2 30024.053} C_VEL
LIN {X 0,Y 679.951,Z 367.94,A -85,B 0,C 180,E1 30023.596,E2 30023.596} C_VEL
LIN {X 0,Y 682.551,Z 372.946,A -85,B 0,C 180,E1 30023.29,E2 30023.29} C_VEL
LIN {X 0,Y 683.761,Z 375.108,A -85,B 0,C 180,E1 30023.152,E2 30023.152} C_VEL
LIN {X 0,Y 680.693,Z 579.396,A -85,B 0,C 180,E1 30020.437,E2 30020.437} C_VEL
LIN {X 0,Y 677.597,Z 803.707,A -85,B 0,C 180,E1 30017.544,E2 30017.544} C_VEL
LIN {X 0,Y 676.87,Z 830.943,A -85,B 0,C 180,E1 30017.131,E2 30017.131} C_VEL
LIN {X 0,Y 675.953,Z 855.351,A -85,B 0,C 180,E1 30016.625,E2 30016.625} C_VEL
LIN {X 0,Y 674.678,Z 882.842,A -85,B 0,C 180,E1 30015.885,E2 30015.885} C_VEL
LIN {X 0,Y 673.279,Z 907.795,A -85,B 0,C 180,E1 30015.042,E2 30015.042} C_VEL
LIN {X 0,Y 671.824,Z 931.596,A -85,B 0,C 180,E1 30014.088,E2 30014.088} C_VEL
LIN {X 0,Y 670.097,Z 957.017,A -85,B 0,C 180,E1 30012.891,E2 30012.891} C_VEL
LIN {X 0,Y 668.236,Z 982.08,A -85,B 0,C 180,E1 30011.517,E2 30011.517} C_VEL
LIN {X 0,Y 666.339,Z 1007.377,A -85,B 0,C 180,E1 30009.907,E2 30009.907} C_VEL
LIN {X 0,Y 664.524,Z 1030.825,A -85,B 0,C 180,E1 30008.199,E2 30008.199} C_VEL
LIN {X 0,Y 662.817,Z 1053.262,A -85,B 0,C 180,E1 30006.335,E2 30006.335} C_VEL
LIN {X 0,Y 661.349,Z 1073.473,A -85,B 0,C 180,E1 30004.432,E2 30004.432} C_VEL
LIN {X 0,Y 659.986,Z 1093.226,A -85,B 0,C 180,E1 30002.329,E2 30002.329} C_VEL
LIN {X 0,Y 658.887,Z 1110.435,A -85,B 0,C 180,E1 30000.252,E2 30000.252} C_VEL
LIN {X 0,Y 657.961,Z 1126.868,A -85,B 0,C 180,E1 29998.001,E2 29998.001} C_VEL
LIN {X 0,Y 657.21,Z 1142.102,A -85,B 0,C 180,E1 29995.599,E2 29995.599} C_VEL
LIN {X 0,Y 656.699,Z 1154.542,A -85,B 0,C 180,E1 29993.32,E2 29993.32} C_VEL
LIN {X 0,Y 656.365,Z 1165.1,A -85,B 0,C 180,E1 29991.07,E2 29991.07} C_VEL
LIN {X 0,Y 656.13,Z 1174.878,A -85,B 0,C 180,E1 29988.572,E2 29988.572} C_VEL
LIN {X 0,Y 656.006,Z 1182.021,A -85,B 0,C 180,E1 29986.287,E2 29986.287} C_VEL
LIN {X 0,Y 655.942,Z 1187.579,A -85,B 0,C 180,E1 29984.026,E2 29984.026} C_VEL
LIN {X 0,Y 655.912,Z 1191.78,A -85,B 0,C 180,E1 29981.608,E2 29981.608} C_VEL
LIN {X 0,Y 655.91,Z 1194.093,A -85,B 0,C 180,E1 29979.387,E2 29979.387} C_VEL
LIN {X 0,Y 655.917,Z 1194.996,A -85,B 0,C 180,E1 29976.917,E2 29976.917} C_VEL
LIN {X 0,Y 655.908,Z 1194.111,A -85,B 0,C 180,E1 29974.547,E2 29974.547} C_VEL
LIN {X 0,Y 655.918,Z 1191.857,A -85,B 0,C 180,E1 29972.359,E2 29972.359} C_VEL
LIN {X 0,Y 655.95,Z 1187.643,A -85,B 0,C 180,E1 29969.913,E2 29969.913} C_VEL
LIN {X 0,Y 656.005,Z 1182.072,A -85,B 0,C 180,E1 29967.642,E2 29967.642} C_VEL
LIN {X 0,Y 656.122,Z 1174.803,A -85,B 0,C 180,E1 29965.317,E2 29965.317} C_VEL
LIN {X 0,Y 656.35,Z 1165.032,A -85,B 0,C 180,E1 29962.824,E2 29962.824} C_VEL
LIN {X 0,Y 656.683,Z 1154.714,A -85,B 0,C 180,E1 29960.624,E2 29960.624} C_VEL
LIN {X 0,Y 657.174,Z 1142.692,A -85,B 0,C 180,E1 29958.414,E2 29958.414} C_VEL
LIN {X 0,Y 657.872,Z 1128.198,A -85,B 0,C 180,E1 29956.106,E2 29956.106} C_VEL
LIN {X 0,Y 658.715,Z 1112.777,A -85,B 0,C 180,E1 29953.963,E2 29953.963} C_VEL
LIN {X 0,Y 659.806,Z 1096.004,A -85,B 0,C 180,E1 29951.901,E2 29951.901} C_VEL
LIN {X 0,Y 661.008,Z 1077.826,A -85,B 0,C 180,E1 29949.918,E2 29949.918} C_VEL
LIN {X 0,Y 662.493,Z 1057.688,A -85,B 0,C 180,E1 29947.973,E2 29947.973} C_VEL
LIN {X 0,Y 664.124,Z 1035.872,A -85,B 0,C 180,E1 29946.11,E2 29946.11} C_VEL
LIN {X 0,Y 665.873,Z 1013.459,A -85,B 0,C 180,E1 29944.424,E2 29944.424} C_VEL
LIN {X 0,Y 667.718,Z 989.237,A -85,B 0,C 180,E1 29942.825,E2 29942.825} C_VEL
LIN {X 0,Y 669.541,Z 964.197,A -85,B 0,C 180,E1 29941.391,E2 29941.391} C_VEL
LIN {X 0,Y 671.386,Z 938.393,A -85,B 0,C 180,E1 29940.122,E2 29940.122} C_VEL
LIN {X 0,Y 673.039,Z 912.423,A -85,B 0,C 180,E1 29939.041,E2 29939.041} C_VEL
LIN {X 0,Y 674.299,Z 889.53,A -85,B 0,C 180,E1 29938.238,E2 29938.238} C_VEL
LIN {X 0,Y 675.523,Z 865.523,A -85,B 0,C 180,E1 29937.539,E2 29937.539} C_VEL
LIN {X 0,Y 676.658,Z 837.332,A -85,B 0,C 180,E1 29936.896,E2 29936.896} C_VEL
LIN {X 0,Y 677.407,Z 812.223,A -85,B 0,C 180,E1 29936.481,E2 29936.481} C_VEL
LIN {X 0,Y 680.489,Z 593.725,A -85,B 0,C 180,E1 29933.66,E2 29933.66} C_VEL
LIN {X 0,Y 683.642,Z 382.304,A -85,B 0,C 180,E1 29930.854,E2 29930.854} C_VEL
LIN {X 0,Y 683.629,Z 374.673,A -85,B 0,C 180,E1 29930.74,E2 29930.74} C_VEL
LIN {X 0,Y 667.77,Z 351.195,A -85,B 0,C 180,E1 29928.931,E2 29928.931} C_VEL
LIN {X 0,Y 660.813,Z 341.43,A -85,B 0,C 180,E1 29928.096,E2 29928.096} C_VEL
LIN {X 0,Y 658.378,Z 336.503,A -85,B 0,C 180,E1 29927.441,E2 29927.441} C_VEL
LIN {X 0,Y 656.705,Z 333.037,A -85,B 0,C 180,E1 29926.957,E2 29926.957} C_VEL
LIN {X 0,Y 656.608,Z 332.446,A -85,B 0,C 180,E1 29926.865,E2 29926.865} C_VEL
LIN {X 0,Y 656.643,Z 332.439,A -85,B 0,C 180,E1 29924.178,E2 29924.178} C_VEL
LIN {X 0,Y 656.619,Z 332.435,A -85,B 0,C 180,E1 29921.02,E2 29921.02} C_VEL
LIN {X 0,Y 656.609,Z 332.438,A -85,B 0,C 180,E1 29918.492,E2 29918.492} C_VEL
LIN {X 0,Y 656.697,Z 332.432,A -85,B 0,C 180,E1 29915.566,E2 29915.566} C_VEL
LIN {X 0,Y 656.611,Z 332.434,A -85,B 0,C 180,E1 29912.621,E2 29912.621} C_VEL
LIN {X 0,Y 656.624,Z 332.437,A -85,B 0,C 180,E1 29910.066,E2 29910.066} C_VEL
LIN {X 0,Y 656.658,Z 332.412,A -85,B 0,C 180,E1 29906.986,E2 29906.986} C_VEL
LIN {X 0,Y 656.612,Z 332.435,A -85,B 0,C 180,E1 29904.278,E2 29904.278} C_VEL
LIN {X 0,Y 656.64,Z 332.403,A -85,B 0,C 180,E1 29901.623,E2 29901.623} C_VEL
LIN {X 0,Y 656.628,Z 332.434,A -85,B 0,C 180,E1 29898.441,E2 29898.441} C_VEL
LIN {X 0,Y 656.614,Z 332.431,A -85,B 0,C 180,E1 29895.909,E2 29895.909} C_VEL
LIN {X 0,Y 656.697,Z 332.425,A -85,B 0,C 180,E1 29893.023,E2 29893.023} C_VEL
LIN {X 0,Y 656.62,Z 332.427,A -85,B 0,C 180,E1 29890.086,E2 29890.086} C_VEL
LIN {X 0,Y 656.624,Z 332.435,A -85,B 0,C 180,E1 29887.525,E2 29887.525} C_VEL
LIN {X 0,Y 656.689,Z 332.432,A -85,B 0,C 180,E1 29884.541,E2 29884.541} C_VEL
LIN {X 0,Y 656.618,Z 332.432,A -85,B 0,C 180,E1 29881.745,E2 29881.745} C_VEL
LIN {X 0,Y 656.631,Z 332.431,A -85,B 0,C 180,E1 29879.215,E2 29879.215} C_VEL
LIN {X 0,Y 656.656,Z 332.424,A -85,B 0,C 180,E1 29876.071,E2 29876.071} C_VEL
LIN {X 0,Y 656.621,Z 332.434,A -85,B 0,C 180,E1 29873.354,E2 29873.354} C_VEL
LIN {X 0,Y 656.686,Z 332.433,A -85,B 0,C 180,E1 29870.535,E2 29870.535} C_VEL
LIN {X 0,Y 656.625,Z 332.404,A -85,B 0,C 180,E1 29867.512,E2 29867.512} C_VEL
LIN {X 0,Y 656.629,Z 332.429,A -85,B 0,C 180,E1 29864.907,E2 29864.907} C_VEL
LIN {X 0,Y 656.686,Z 332.406,A -85,B 0,C 180,E1 29861.904,E2 29861.904} C_VEL
LIN {X 0,Y 656.625,Z 332.429,A -85,B 0,C 180,E1 29859.125,E2 29859.125} C_VEL
LIN {X 0,Y 656.637,Z 332.427,A -85,B 0,C 180,E1 29856.582,E2 29856.582} C_VEL
LIN {X 0,Y 656.649,Z 332.433,A -85,B 0,C 180,E1 29853.355,E2 29853.355} C_VEL
LIN {X 0,Y 656.627,Z 332.433,A -85,B 0,C 180,E1 29850.738,E2 29850.738} C_VEL
LIN {X 0,Y 656.705,Z 332.432,A -85,B 0,C 180,E1 29847.836,E2 29847.836} C_VEL
LIN {X 0,Y 656.633,Z 332.436,A -85,B 0,C 180,E1 29844.854,E2 29844.854} C_VEL
LIN {X 0,Y 656.649,Z 332.438,A -85,B 0,C 180,E1 29842.146,E2 29842.146} C_VEL
LIN {X 0,Y 656.648,Z 332.525,A -85,B 0,C 180,E1 29840.836,E2 29840.836} C_VEL
LIN {X 0,Y 657.986,Z 336,A -85,B 0,C 180,E1 29840.392,E2 29840.392} C_VEL
LIN {X 0,Y 659.124,Z 338.218,A -85,B 0,C 180,E1 29840.082,E2 29840.082} C_VEL
LIN {X 0,Y 661.381,Z 342.902,A -85,B 0,C 180,E1 29839.452,E2 29839.452} C_VEL
LIN {X 0,Y 665.398,Z 351.071,A -85,B 0,C 180,E1 29838.408,E2 29838.408} C_VEL
LIN {X 0,Y 681.166,Z 373.894,A -85,B 0,C 180,E1 29836.594,E2 29836.594} C_VEL
LIN {X 0,Y 683.516,Z 378.011,A -85,B 0,C 180,E1 29836.324,E2 29836.324} C_VEL
LIN {X 0,Y 683.819,Z 380.637,A -85,B 0,C 180,E1 29836.259,E2 29836.259} C_VEL
LIN {X 0,Y 680.667,Z 591.291,A -85,B 0,C 180,E1 29833.457,E2 29833.457} C_VEL
LIN {X 0,Y 677.589,Z 814.102,A -85,B 0,C 180,E1 29830.584,E2 29830.584} C_VEL
LIN {X 0,Y 676.833,Z 842.087,A -85,B 0,C 180,E1 29830.156,E2 29830.156} C_VEL
LIN {X 0,Y 675.92,Z 865.96,A -85,B 0,C 180,E1 29829.655,E2 29829.655} C_VEL
LIN {X 0,Y 674.726,Z 891.895,A -85,B 0,C 180,E1 29828.96,E2 29828.96} C_VEL
LIN {X 0,Y 673.228,Z 918.756,A -85,B 0,C 180,E1 29828.05,E2 29828.05} C_VEL
LIN {X 0,Y 671.9,Z 939.842,A -85,B 0,C 180,E1 29827.206,E2 29827.206} C_VEL
LIN {X 0,Y 670.501,Z 960.729,A -85,B 0,C 180,E1 29826.247,E2 29826.247} C_VEL
LIN {X 0,Y 668.872,Z 983.908,A -85,B 0,C 180,E1 29825.031,E2 29825.031} C_VEL
LIN {X 0,Y 666.982,Z 1008.529,A -85,B 0,C 180,E1 29823.538,E2 29823.538} C_VEL
LIN {X 0,Y 665.451,Z 1028.186,A -85,B 0,C 180,E1 29822.189,E2 29822.189} C_VEL
LIN {X 0,Y 663.951,Z 1048.296,A -85,B 0,C 180,E1 29820.647,E2 29820.647} C_VEL
LIN {X 0,Y 662.313,Z 1070.05,A -85,B 0,C 180,E1 29818.76,E2 29818.76} C_VEL
LIN {X 0,Y 661.057,Z 1086.854,A -85,B 0,C 180,E1 29817.131,E2 29817.131} C_VEL
LIN {X 0,Y 659.907,Z 1104.463,A -85,B 0,C 180,E1 29815.233,E2 29815.233} C_VEL
LIN {X 0,Y 658.773,Z 1121.891,A -85,B 0,C 180,E1 29813.104,E2 29813.104} C_VEL
LIN {X 0,Y 658.001,Z 1135.754,A -85,B 0,C 180,E1 29811.201,E2 29811.201} C_VEL
LIN {X 0,Y 657.305,Z 1150.032,A -85,B 0,C 180,E1 29808.997,E2 29808.997} C_VEL
LIN {X 0,Y 656.751,Z 1162.679,A -85,B 0,C 180,E1 29806.723,E2 29806.723} C_VEL
LIN {X 0,Y 656.451,Z 1171.896,A -85,B 0,C 180,E1 29804.826,E2 29804.826} C_VEL
LIN {X 0,Y 656.232,Z 1179.871,A -85,B 0,C 180,E1 29802.943,E2 29802.943} C_VEL
LIN {X 0,Y 656.049,Z 1187.893,A -85,B 0,C 180,E1 29800.716,E2 29800.716} C_VEL
LIN {X 0,Y 655.97,Z 1194.694,A -85,B 0,C 180,E1 29798.326,E2 29798.326} C_VEL
LIN {X 0,Y 655.929,Z 1199.41,A -85,B 0,C 180,E1 29796.125,E2 29796.125} C_VEL
LIN {X 0,Y 655.91,Z 1202.789,A -85,B 0,C 180,E1 29793.846,E2 29793.846} C_VEL
LIN {X 0,Y 655.911,Z 1204.624,A -85,B 0,C 180,E1 29791.485,E2 29791.485} C_VEL
LIN {X 0,Y 655.893,Z 1204.849,A -85,B 0,C 180,E1 29789.389,E2 29789.389} C_VEL
LIN {X 0,Y 655.908,Z 1203.947,A -85,B 0,C 180,E1 29787.379,E2 29787.379} C_VEL
LIN {X 0,Y 655.919,Z 1201.428,A -85,B 0,C 180,E1 29785.103,E2 29785.103} C_VEL
LIN {X 0,Y 655.949,Z 1197.152,A -85,B 0,C 180,E1 29782.732,E2 29782.732} C_VEL
LIN {X 0,Y 656.009,Z 1191.376,A -85,B 0,C 180,E1 29780.437,E2 29780.437} C_VEL
LIN {X 0,Y 656.126,Z 1184.279,A -85,B 0,C 180,E1 29778.217,E2 29778.217} C_VEL
LIN {X 0,Y 656.39,Z 1174.089,A -85,B 0,C 180,E1 29775.658,E2 29775.658} C_VEL
LIN {X 0,Y 656.692,Z 1164.276,A -85,B 0,C 180,E1 29773.588,E2 29773.588} C_VEL
LIN {X 0,Y 657.112,Z 1154.137,A -85,B 0,C 180,E1 29771.716,E2 29771.716} C_VEL
LIN {X 0,Y 657.764,Z 1140.78,A -85,B 0,C 180,E1 29769.536,E2 29769.536} C_VEL
LIN {X 0,Y 658.6,Z 1125.104,A -85,B 0,C 180,E1 29767.318,E2 29767.318} C_VEL
LIN {X 0,Y 659.476,Z 1110.399,A -85,B 0,C 180,E1 29765.467,E2 29765.467} C_VEL
LIN {X 0,Y 660.73,Z 1092.313,A -85,B 0,C 180,E1 29763.428,E2 29763.428} C_VEL
LIN {X 0,Y 662,Z 1073.819,A -85,B 0,C 180,E1 29761.591,E2 29761.591} C_VEL
LIN {X 0,Y 663.289,Z 1056.842,A -85,B 0,C 180,E1 29760.069,E2 29760.069} C_VEL
LIN {X 0,Y 664.962,Z 1035.53,A -85,B 0,C 180,E1 29758.348,E2 29758.348} C_VEL
LIN {X 0,Y 666.618,Z 1013.003,A -85,B 0,C 180,E1 29756.756,E2 29756.756} C_VEL
LIN {X 0,Y 668.131,Z 993.022,A -85,B 0,C 180,E1 29755.499,E2 29755.499} C_VEL
LIN {X 0,Y 669.972,Z 968.967,A -85,B 0,C 180,E1 29754.161,E2 29754.161} C_VEL
LIN {X 0,Y 671.657,Z 944.001,A -85,B 0,C 180,E1 29752.976,E2 29752.976} C_VEL
LIN {X 0,Y 672.974,Z 923.056,A -85,B 0,C 180,E1 29752.114,E2 29752.114} C_VEL
LIN {X 0,Y 674.098,Z 902.837,A -85,B 0,C 180,E1 29751.392,E2 29751.392} C_VEL
LIN {X 0,Y 675.318,Z 879.538,A -85,B 0,C 180,E1 29750.689,E2 29750.689} C_VEL
LIN {X 0,Y 676.525,Z 851.649,A -85,B 0,C 180,E1 29750.026,E2 29750.026} C_VEL
LIN {X 0,Y 677.299,Z 826.243,A -85,B 0,C 180,E1 29749.585,E2 29749.585} C_VEL
LIN {X 0,Y 680.398,Z 610.206,A -85,B 0,C 180,E1 29746.79,E2 29746.79} C_VEL
LIN {X 0,Y 683.424,Z 405.953,A -85,B 0,C 180,E1 29744.083,E2 29744.083} C_VEL
LIN {X 0,Y 683.694,Z 378.682,A -85,B 0,C 180,E1 29743.701,E2 29743.701} C_VEL
LIN {X 0,Y 682.678,Z 376.226,A -85,B 0,C 180,E1 29743.575,E2 29743.575} C_VEL
LIN {X 0,Y 669.174,Z 356.394,A -85,B 0,C 180,E1 29742.038,E2 29742.038} C_VEL
LIN {X 0,Y 664.949,Z 350.19,A -85,B 0,C 180,E1 29741.512,E2 29741.512} C_VEL
LIN {X 0,Y 660.092,Z 340.16,A -85,B 0,C 180,E1 29740.188,E2 29740.188} C_VEL
LIN {X 0,Y 658.152,Z 336.22,A -85,B 0,C 180,E1 29739.649,E2 29739.649} C_VEL
LIN {X 0,Y 656.682,Z 332.733,A -85,B 0,C 180,E1 29739.19,E2 29739.19} C_VEL
LIN {X 0,Y 656.648,Z 332.44,A -85,B 0,C 180,E1 29739.053,E2 29739.053} C_VEL
LIN {X 0,Y 656.667,Z 332.432,A -85,B 0,C 180,E1 29735.89,E2 29735.89} C_VEL
LIN {X 0,Y 656.637,Z 332.434,A -85,B 0,C 180,E1 29733.125,E2 29733.125} C_VEL
LIN {X 0,Y 656.715,Z 332.414,A -85,B 0,C 180,E1 29730.142,E2 29730.142} C_VEL
LIN {X 0,Y 656.634,Z 332.409,A -85,B 0,C 180,E1 29727.183,E2 29727.183} C_VEL
LIN {X 0,Y 656.679,Z 332.431,A -85,B 0,C 180,E1 29724.371,E2 29724.371} C_VEL
LIN {X 0,Y 656.649,Z 332.425,A -85,B 0,C 180,E1 29721.248,E2 29721.248} C_VEL
LIN {X 0,Y 656.646,Z 332.425,A -85,B 0,C 180,E1 29718.557,E2 29718.557} C_VEL
LIN {X 0,Y 656.692,Z 332.429,A -85,B 0,C 180,E1 29715.454,E2 29715.454} C_VEL
LIN {X 0,Y 656.638,Z 332.411,A -85,B 0,C 180,E1 29712.667,E2 29712.667} C_VEL
LIN {X 0,Y 656.706,Z 332.426,A -85,B 0,C 180,E1 29709.73,E2 29709.73} C_VEL
LIN {X 0,Y 656.644,Z 332.409,A -85,B 0,C 180,E1 29706.733,E2 29706.733} C_VEL
LIN {X 0,Y 656.658,Z 332.43,A -85,B 0,C 180,E1 29704.017,E2 29704.017} C_VEL
LIN {X 0,Y 656.664,Z 332.411,A -85,B 0,C 180,E1 29700.785,E2 29700.785} C_VEL
LIN {X 0,Y 656.645,Z 332.431,A -85,B 0,C 180,E1 29698.08,E2 29698.08} C_VEL
LIN {X 0,Y 656.706,Z 332.405,A -85,B 0,C 180,E1 29695.021,E2 29695.021} C_VEL
LIN {X 0,Y 656.644,Z 332.427,A -85,B 0,C 180,E1 29692.123,E2 29692.123} C_VEL
LIN {X 0,Y 656.7,Z 332.413,A -85,B 0,C 180,E1 29689.206,E2 29689.206} C_VEL
LIN {X 0,Y 656.65,Z 332.413,A -85,B 0,C 180,E1 29686.168,E2 29686.168} C_VEL
LIN {X 0,Y 656.668,Z 332.428,A -85,B 0,C 180,E1 29683.366,E2 29683.366} C_VEL
LIN {X 0,Y 656.665,Z 332.414,A -85,B 0,C 180,E1 29680.15,E2 29680.15} C_VEL
LIN {X 0,Y 656.652,Z 332.427,A -85,B 0,C 180,E1 29677.435,E2 29677.435} C_VEL
LIN {X 0,Y 656.706,Z 332.431,A -85,B 0,C 180,E1 29674.334,E2 29674.334} C_VEL
LIN {X 0,Y 656.65,Z 332.435,A -85,B 0,C 180,E1 29671.436,E2 29671.436} C_VEL
LIN {X 0,Y 656.713,Z 332.428,A -85,B 0,C 180,E1 29668.496,E2 29668.496} C_VEL
LIN {X 0,Y 656.682,Z 332.581,A -85,B 0,C 180,E1 29667,E2 29667} C_VEL
LIN {X 0,Y 658.15,Z 336.115,A -85,B 0,C 180,E1 29666.531,E2 29666.531} C_VEL
LIN {X 0,Y 659.206,Z 338.39,A -85,B 0,C 180,E1 29666.22,E2 29666.22} C_VEL
LIN {X 0,Y 660.909,Z 341.551,A -85,B 0,C 180,E1 29665.803,E2 29665.803} C_VEL
LIN {X 0,Y 664.254,Z 346.197,A -85,B 0,C 180,E1 29665.398,E2 29665.398} C_VEL
LIN {X 0,Y 680.642,Z 370.02,A -85,B 0,C 180,E1 29663.503,E2 29663.503} C_VEL
LIN {X 0,Y 682.551,Z 372.946,A -85,B 0,C 180,E1 29663.29,E2 29663.29} C_VEL
LIN {X 0,Y 683.268,Z 375.244,A -85,B 0,C 180,E1 29663.193,E2 29663.193} C_VEL
LIN {X 0,Y 682.927,Z 379.457,A -85,B 0,C 180,E1 29663.16,E2 29663.16} C_VEL
LIN {X 0,Y 680.704,Z 386.055,A -85,B 0,C 180,E1 29663.257,E2 29663.257} C_VEL
LIN {X 0,Y 678.263,Z 393.171,A -85,B 0,C 180,E1 29663.366,E2 29663.366} C_VEL
LIN {X 0,Y 677.843,Z 396.468,A -85,B 0,C 180,E1 29663.354,E2 29663.354} C_VEL
LIN {X 0,Y 674.579,Z 599.09,A -85,B 0,C 180,E1 29660.647,E2 29660.647} C_VEL
LIN {X 0,Y 671.219,Z 816.142,A -85,B 0,C 180,E1 29657.817,E2 29657.817} C_VEL
LIN {X 0,Y 670.288,Z 843.874,A -85,B 0,C 180,E1 29657.325,E2 29657.325} C_VEL
LIN {X 0,Y 669.098,Z 868.751,A -85,B 0,C 180,E1 29656.725,E2 29656.725} C_VEL
LIN {X 0,Y 667.831,Z 892.094,A -85,B 0,C 180,E1 29656.025,E2 29656.025} C_VEL
LIN {X 0,Y 666.272,Z 917.665,A -85,B 0,C 180,E1 29655.098,E2 29655.098} C_VEL
LIN {X 0,Y 664.457,Z 942.886,A -85,B 0,C 180,E1 29654.003,E2 29654.003} C_VEL
LIN {X 0,Y 662.641,Z 966.649,A -85,B 0,C 180,E1 29652.803,E2 29652.803} C_VEL
LIN {X 0,Y 660.655,Z 991.448,A -85,B 0,C 180,E1 29651.35,E2 29651.35} C_VEL
LIN {X 0,Y 658.721,Z 1014.887,A -85,B 0,C 180,E1 29649.776,E2 29649.776} C_VEL
LIN {X 0,Y 656.722,Z 1038.526,A -85,B 0,C 180,E1 29647.958,E2 29647.958} C_VEL
LIN {X 0,Y 654.995,Z 1059.763,A -85,B 0,C 180,E1 29646.103,E2 29646.103} C_VEL
LIN {X 0,Y 653.344,Z 1080.347,A -85,B 0,C 180,E1 29644.064,E2 29644.064} C_VEL
LIN {X 0,Y 651.966,Z 1099.195,A -85,B 0,C 180,E1 29641.944,E2 29641.944} C_VEL
LIN {X 0,Y 650.814,Z 1116.416,A -85,B 0,C 180,E1 29639.751,E2 29639.751} C_VEL
LIN {X 0,Y 649.849,Z 1132.602,A -85,B 0,C 180,E1 29637.39,E2 29637.39} C_VEL
LIN {X 0,Y 649.131,Z 1146.478,A -85,B 0,C 180,E1 29635.061,E2 29635.061} C_VEL
LIN {X 0,Y 648.62,Z 1158.759,A -85,B 0,C 180,E1 29632.667,E2 29632.667} C_VEL
LIN {X 0,Y 648.29,Z 1168.927,A -85,B 0,C 180,E1 29630.305,E2 29630.305} C_VEL
LIN {X 0,Y 648.09,Z 1176.714,A -85,B 0,C 180,E1 29628.158,E2 29628.158} C_VEL
LIN {X 0,Y 647.99,Z 1183.28,A -85,B 0,C 180,E1 29625.942,E2 29625.942} C_VEL
LIN {X 0,Y 647.937,Z 1188.845,A -85,B 0,C 180,E1 29623.475,E2 29623.475} C_VEL
LIN {X 0,Y 647.916,Z 1192.347,A -85,B 0,C 180,E1 29621.212,E2 29621.212} C_VEL
LIN {X 0,Y 647.909,Z 1194.45,A -85,B 0,C 180,E1 29618.877,E2 29618.877} C_VEL
LIN {X 0,Y 647.905,Z 1194.885,A -85,B 0,C 180,E1 29616.468,E2 29616.468} C_VEL
LIN {X 0,Y 647.909,Z 1193.973,A -85,B 0,C 180,E1 29614.337,E2 29614.337} C_VEL
LIN {X 0,Y 647.922,Z 1191.485,A -85,B 0,C 180,E1 29612.034,E2 29612.034} C_VEL
LIN {X 0,Y 647.948,Z 1187.175,A -85,B 0,C 180,E1 29609.612,E2 29609.612} C_VEL
LIN {X 0,Y 648.017,Z 1181.577,A -85,B 0,C 180,E1 29607.347,E2 29607.347} C_VEL
LIN {X 0,Y 648.148,Z 1174.353,A -85,B 0,C 180,E1 29605.044,E2 29605.044} C_VEL
LIN {X 0,Y 648.431,Z 1164.538,A -85,B 0,C 180,E1 29602.534,E2 29602.534} C_VEL
LIN {X 0,Y 648.796,Z 1154.263,A -85,B 0,C 180,E1 29600.33,E2 29600.33} C_VEL
LIN {X 0,Y 649.379,Z 1141.683,A -85,B 0,C 180,E1 29598.003,E2 29598.003} C_VEL
LIN {X 0,Y 650.2,Z 1126.387,A -85,B 0,C 180,E1 29595.575,E2 29595.575} C_VEL
LIN {X 0,Y 651.228,Z 1110.052,A -85,B 0,C 180,E1 29593.315,E2 29593.315} C_VEL
LIN {X 0,Y 652.517,Z 1091.298,A -85,B 0,C 180,E1 29591.044,E2 29591.044} C_VEL
LIN {X 0,Y 653.977,Z 1072.484,A -85,B 0,C 180,E1 29589.037,E2 29589.037} C_VEL
LIN {X 0,Y 655.683,Z 1051.106,A -85,B 0,C 180,E1 29587.022,E2 29587.022} C_VEL
LIN {X 0,Y 657.539,Z 1028.93,A -85,B 0,C 180,E1 29585.185,E2 29585.185} C_VEL
LIN {X 0,Y 659.473,Z 1005.563,A -85,B 0,C 180,E1 29583.48,E2 29583.48} C_VEL
LIN {X 0,Y 661.523,Z 980.827,A -85,B 0,C 180,E1 29581.913,E2 29581.913} C_VEL
LIN {X 0,Y 663.465,Z 956.513,A -85,B 0,C 180,E1 29580.575,E2 29580.575} C_VEL
LIN {X 0,Y 665.383,Z 930.046,A -85,B 0,C 180,E1 29579.326,E2 29579.326} C_VEL
LIN {X 0,Y 666.989,Z 905.63,A -85,B 0,C 180,E1 29578.354,E2 29578.354} C_VEL
LIN {X 0,Y 668.622,Z 878.756,A -85,B 0,C 180,E1 29577.464,E2 29577.464} C_VEL
LIN {X 0,Y 669.845,Z 853.126,A -85,B 0,C 180,E1 29576.793,E2 29576.793} C_VEL
LIN {X 0,Y 670.809,Z 828.841,A -85,B 0,C 180,E1 29576.297,E2 29576.297} C_VEL
LIN {X 0,Y 671.612,Z 797.294,A -85,B 0,C 180,E1 29575.838,E2 29575.838} C_VEL
LIN {X 0,Y 674.96,Z 574.803,A -85,B 0,C 180,E1 29572.943,E2 29572.943} C_VEL
LIN {X 0,Y 678.155,Z 378.612,A -85,B 0,C 180,E1 29570.315,E2 29570.315} C_VEL
LIN {X 0,Y 663.295,Z 356.724,A -85,B 0,C 180,E1 29568.587,E2 29568.587} C_VEL
LIN {X 0,Y 652.308,Z 341.469,A -85,B 0,C 180,E1 29567.232,E2 29567.232} C_VEL
LIN {X 0,Y 650.275,Z 337.332,A -85,B 0,C 180,E1 29566.661,E2 29566.661} C_VEL
LIN {X 0,Y 648.841,Z 334.208,A -85,B 0,C 180,E1 29566.219,E2 29566.219} C_VEL
LIN {X 0,Y 648.723,Z 333.432,A -85,B 0,C 180,E1 29566.087,E2 29566.087} C_VEL
LIN {X 0,Y 648.679,Z 333.415,A -85,B 0,C 180,E1 29563.063,E2 29563.063} C_VEL
LIN {X 0,Y 648.674,Z 333.428,A -85,B 0,C 180,E1 29560.462,E2 29560.462} C_VEL
LIN {X 0,Y 648.748,Z 333.418,A -85,B 0,C 180,E1 29557.465,E2 29557.465} C_VEL
LIN {X 0,Y 648.67,Z 333.419,A -85,B 0,C 180,E1 29554.559,E2 29554.559} C_VEL
LIN {X 0,Y 648.711,Z 333.419,A -85,B 0,C 180,E1 29551.813,E2 29551.813} C_VEL
LIN {X 0,Y 648.685,Z 333.402,A -85,B 0,C 180,E1 29548.714,E2 29548.714} C_VEL
LIN {X 0,Y 648.674,Z 333.416,A -85,B 0,C 180,E1 29546.158,E2 29546.158} C_VEL
LIN {X 0,Y 648.761,Z 333.401,A -85,B 0,C 180,E1 29543.238,E2 29543.238} C_VEL
LIN {X 0,Y 648.676,Z 333.412,A -85,B 0,C 180,E1 29540.293,E2 29540.293} C_VEL
LIN {X 0,Y 648.691,Z 333.425,A -85,B 0,C 180,E1 29537.677,E2 29537.677} C_VEL
LIN {X 0,Y 648.7,Z 333.42,A -85,B 0,C 180,E1 29534.46,E2 29534.46} C_VEL
LIN {X 0,Y 648.676,Z 333.424,A -85,B 0,C 180,E1 29531.826,E2 29531.826} C_VEL
LIN {X 0,Y 648.763,Z 333.415,A -85,B 0,C 180,E1 29528.866,E2 29528.866} C_VEL
LIN {X 0,Y 648.681,Z 333.417,A -85,B 0,C 180,E1 29525.928,E2 29525.928} C_VEL
LIN {X 0,Y 648.695,Z 333.424,A -85,B 0,C 180,E1 29523.269,E2 29523.269} C_VEL
LIN {X 0,Y 648.698,Z 333.418,A -85,B 0,C 180,E1 29520,E2 29520} C_VEL
LIN {X 0,Y 648.683,Z 333.424,A -85,B 0,C 180,E1 29517.35,E2 29517.35} C_VEL
LIN {X 0,Y 648.762,Z 333.421,A -85,B 0,C 180,E1 29514.339,E2 29514.339} C_VEL
LIN {X 0,Y 648.683,Z 333.419,A -85,B 0,C 180,E1 29511.49,E2 29511.49} C_VEL
LIN {X 0,Y 648.706,Z 333.414,A -85,B 0,C 180,E1 29508.801,E2 29508.801} C_VEL
LIN {X 0,Y 648.703,Z 333.412,A -85,B 0,C 180,E1 29505.631,E2 29505.631} C_VEL
LIN {X 0,Y 648.685,Z 333.423,A -85,B 0,C 180,E1 29503.063,E2 29503.063} C_VEL
LIN {X 0,Y 648.769,Z 333.389,A -85,B 0,C 180,E1 29500.069,E2 29500.069} C_VEL
LIN {X 0,Y 648.687,Z 333.42,A -85,B 0,C 180,E1 29497.143,E2 29497.143} C_VEL
LIN {X 0,Y 648.698,Z 333.394,A -85,B 0,C 180,E1 29494.529,E2 29494.529} C_VEL
LIN {X 0,Y 648.716,Z 333.417,A -85,B 0,C 180,E1 29491.357,E2 29491.357} C_VEL
LIN {X 0,Y 648.688,Z 333.42,A -85,B 0,C 180,E1 29488.704,E2 29488.704} C_VEL
LIN {X 0,Y 648.768,Z 333.421,A -85,B 0,C 180,E1 29485.768,E2 29485.768} C_VEL
LIN {X 0,Y 648.697,Z 333.427,A -85,B 0,C 180,E1 29482.827,E2 29482.827} C_VEL
LIN {X 0,Y 648.776,Z 333.443,A -85,B 0,C 180,E1 29481.603,E2 29481.603} C_VEL
LIN {X 0,Y 650.118,Z 337.037,A -85,B 0,C 180,E1 29481.133,E2 29481.133} C_VEL
LIN {X 0,Y 651.114,Z 339.025,A -85,B 0,C 180,E1 29480.849,E2 29480.849} C_VEL
LIN {X 0,Y 655.704,Z 348.501,A -85,B 0,C 180,E1 29479.544,E2 29479.544} C_VEL
LIN {X 0,Y 657.153,Z 351.107,A -85,B 0,C 180,E1 29479.222,E2 29479.222} C_VEL
LIN {X 0,Y 674.402,Z 375.96,A -85,B 0,C 180,E1 29477.173,E2 29477.173} C_VEL
LIN {X 0,Y 678.258,Z 382.034,A -85,B 0,C 180,E1 29476.731,E2 29476.731} C_VEL
LIN {X 0,Y 674.838,Z 592.41,A -85,B 0,C 180,E1 29473.912,E2 29473.912} C_VEL
LIN {X 0,Y 671.488,Z 815.507,A -85,B 0,C 180,E1 29471.012,E2 29471.012} C_VEL
LIN {X 0,Y 670.667,Z 842.874,A -85,B 0,C 180,E1 29470.584,E2 29470.584} C_VEL
LIN {X 0,Y 669.702,Z 866.331,A -85,B 0,C 180,E1 29470.086,E2 29470.086} C_VEL
LIN {X 0,Y 668.407,Z 892.412,A -85,B 0,C 180,E1 29469.382,E2 29469.382} C_VEL
LIN {X 0,Y 666.802,Z 918.753,A -85,B 0,C 180,E1 29468.483,E2 29468.483} C_VEL
LIN {X 0,Y 665.363,Z 939.923,A -85,B 0,C 180,E1 29467.63,E2 29467.63} C_VEL
LIN {X 0,Y 663.854,Z 960.724,A -85,B 0,C 180,E1 29466.668,E2 29466.668} C_VEL
LIN {X 0,Y 662.096,Z 983.911,A -85,B 0,C 180,E1 29465.443,E2 29465.443} C_VEL
LIN {X 0,Y 660.054,Z 1008.607,A -85,B 0,C 180,E1 29463.932,E2 29463.932} C_VEL
LIN {X 0,Y 658.45,Z 1027.583,A -85,B 0,C 180,E1 29462.62,E2 29462.62} C_VEL
LIN {X 0,Y 656.822,Z 1047.088,A -85,B 0,C 180,E1 29461.118,E2 29461.118} C_VEL
LIN {X 0,Y 654.983,Z 1069.759,A -85,B 0,C 180,E1 29459.141,E2 29459.141} C_VEL
LIN {X 0,Y 653.646,Z 1086.39,A -85,B 0,C 180,E1 29457.513,E2 29457.513} C_VEL
LIN {X 0,Y 652.369,Z 1103.306,A -85,B 0,C 180,E1 29455.679,E2 29455.679} C_VEL
LIN {X 0,Y 651.106,Z 1121.566,A -85,B 0,C 180,E1 29453.436,E2 29453.436} C_VEL
LIN {X 0,Y 650.244,Z 1135.429,A -85,B 0,C 180,E1 29451.515,E2 29451.515} C_VEL
LIN {X 0,Y 649.487,Z 1149.548,A -85,B 0,C 180,E1 29449.313,E2 29449.313} C_VEL
LIN {X 0,Y 648.875,Z 1162.215,A -85,B 0,C 180,E1 29447.024,E2 29447.024} C_VEL
LIN {X 0,Y 648.512,Z 1171.487,A -85,B 0,C 180,E1 29445.103,E2 29445.103} C_VEL
LIN {X 0,Y 648.281,Z 1179.515,A -85,B 0,C 180,E1 29443.195,E2 29443.195} C_VEL
LIN {X 0,Y 648.084,Z 1187.034,A -85,B 0,C 180,E1 29441.112,E2 29441.112} C_VEL
LIN {X 0,Y 647.987,Z 1193.816,A -85,B 0,C 180,E1 29438.787,E2 29438.787} C_VEL
LIN {X 0,Y 647.935,Z 1199.101,A -85,B 0,C 180,E1 29436.372,E2 29436.372} C_VEL
LIN {X 0,Y 647.918,Z 1202.476,A -85,B 0,C 180,E1 29434.159,E2 29434.159} C_VEL
LIN {X 0,Y 647.907,Z 1204.549,A -85,B 0,C 180,E1 29431.769,E2 29431.769} C_VEL
LIN {X 0,Y 647.892,Z 1204.872,A -85,B 0,C 180,E1 29429.469,E2 29429.469} C_VEL
LIN {X 0,Y 647.909,Z 1203.944,A -85,B 0,C 180,E1 29427.346,E2 29427.346} C_VEL
LIN {X 0,Y 647.922,Z 1201.427,A -85,B 0,C 180,E1 29425.042,E2 29425.042} C_VEL
LIN {X 0,Y 647.951,Z 1197.151,A -85,B 0,C 180,E1 29422.641,E2 29422.641} C_VEL
LIN {X 0,Y 648.018,Z 1191.373,A -85,B 0,C 180,E1 29420.318,E2 29420.318} C_VEL
LIN {X 0,Y 648.146,Z 1184.279,A -85,B 0,C 180,E1 29418.07,E2 29418.07} C_VEL
LIN {X 0,Y 648.439,Z 1174.338,A -85,B 0,C 180,E1 29415.535,E2 29415.535} C_VEL
LIN {X 0,Y 648.769,Z 1164.544,A -85,B 0,C 180,E1 29413.434,E2 29413.434} C_VEL
LIN {X 0,Y 649.238,Z 1154.237,A -85,B 0,C 180,E1 29411.503,E2 29411.503} C_VEL
LIN {X 0,Y 649.924,Z 1141.364,A -85,B 0,C 180,E1 29409.372,E2 29409.372} C_VEL
LIN {X 0,Y 650.838,Z 1125.803,A -85,B 0,C 180,E1 29407.128,E2 29407.128} C_VEL
LIN {X 0,Y 651.804,Z 1111.152,A -85,B 0,C 180,E1 29405.252,E2 29405.252} C_VEL
LIN {X 0,Y 653.113,Z 1093.727,A -85,B 0,C 180,E1 29403.251,E2 29403.251} C_VEL
LIN {X 0,Y 654.547,Z 1074.831,A -85,B 0,C 180,E1 29401.337,E2 29401.337} C_VEL
LIN {X 0,Y 655.937,Z 1057.951,A -85,B 0,C 180,E1 29399.8,E2 29399.8} C_VEL
LIN {X 0,Y 657.511,Z 1039.194,A -85,B 0,C 180,E1 29398.254,E2 29398.254} C_VEL
LIN {X 0,Y 659.486,Z 1015.132,A -85,B 0,C 180,E1 29396.501,E2 29396.501} C_VEL
LIN {X 0,Y 661.142,Z 994.951,A -85,B 0,C 180,E1 29395.207,E2 29395.207} C_VEL
LIN {X 0,Y 662.831,Z 974.061,A -85,B 0,C 180,E1 29394.017,E2 29394.017} C_VEL
LIN {X 0,Y 664.822,Z 948.476,A -85,B 0,C 180,E1 29392.747,E2 29392.747} C_VEL
LIN {X 0,Y 666.407,Z 925.174,A -85,B 0,C 180,E1 29391.764,E2 29391.764} C_VEL
LIN {X 0,Y 667.661,Z 904.465,A -85,B 0,C 180,E1 29391.01,E2 29391.01} C_VEL
LIN {X 0,Y 668.911,Z 882.309,A -85,B 0,C 180,E1 29390.328,E2 29390.328} C_VEL
LIN {X 0,Y 670.161,Z 856.684,A -85,B 0,C 180,E1 29389.689,E2 29389.689} C_VEL
LIN {X 0,Y 671.133,Z 829.115,A -85,B 0,C 180,E1 29389.183,E2 29389.183} C_VEL
LIN {X 0,Y 672.994,Z 712.976,A -85,B 0,C 180,E1 29387.666,E2 29387.666} C_VEL
LIN {X 0,Y 676.404,Z 494.255,A -85,B 0,C 180,E1 29384.784,E2 29384.784} C_VEL
LIN {X 0,Y 678.144,Z 381.612,A -85,B 0,C 180,E1 29383.253,E2 29383.253} C_VEL
LIN {X 0,Y 663.415,Z 359.972,A -85,B 0,C 180,E1 29381.542,E2 29381.542} C_VEL
LIN {X 0,Y 656.505,Z 350.04,A -85,B 0,C 180,E1 29380.672,E2 29380.672} C_VEL
LIN {X 0,Y 652.319,Z 341.504,A -85,B 0,C 180,E1 29379.503,E2 29379.503} C_VEL
LIN {X 0,Y 650.102,Z 337.011,A -85,B 0,C 180,E1 29378.868,E2 29378.868} C_VEL
LIN {X 0,Y 648.774,Z 333.421,A -85,B 0,C 180,E1 29378.364,E2 29378.364} C_VEL
LIN {X 0,Y 648.696,Z 333.427,A -85,B 0,C 180,E1 29375.377,E2 29375.377} C_VEL
LIN {X 0,Y 648.746,Z 333.411,A -85,B 0,C 180,E1 29372.537,E2 29372.537} C_VEL
LIN {X 0,Y 648.707,Z 333.425,A -85,B 0,C 180,E1 29369.444,E2 29369.444} C_VEL
LIN {X 0,Y 648.705,Z 333.396,A -85,B 0,C 180,E1 29366.749,E2 29366.749} C_VEL
LIN {X 0,Y 648.741,Z 333.406,A -85,B 0,C 180,E1 29363.624,E2 29363.624} C_VEL
LIN {X 0,Y 648.699,Z 333.419,A -85,B 0,C 180,E1 29360.858,E2 29360.858} C_VEL
LIN {X 0,Y 648.764,Z 333.395,A -85,B 0,C 180,E1 29357.954,E2 29357.954} C_VEL
LIN {X 0,Y 648.704,Z 333.423,A -85,B 0,C 180,E1 29354.894,E2 29354.894} C_VEL
LIN {X 0,Y 648.729,Z 333.392,A -85,B 0,C 180,E1 29352.1,E2 29352.1} C_VEL
LIN {X 0,Y 648.714,Z 333.419,A -85,B 0,C 180,E1 29348.898,E2 29348.898} C_VEL
LIN {X 0,Y 648.708,Z 333.399,A -85,B 0,C 180,E1 29346.194,E2 29346.194} C_VEL
LIN {X 0,Y 648.752,Z 333.412,A -85,B 0,C 180,E1 29343.092,E2 29343.092} C_VEL
LIN {X 0,Y 648.702,Z 333.41,A -85,B 0,C 180,E1 29340.265,E2 29340.265} C_VEL
LIN {X 0,Y 648.767,Z 333.41,A -85,B 0,C 180,E1 29337.35,E2 29337.35} C_VEL
LIN {X 0,Y 648.709,Z 333.417,A -85,B 0,C 180,E1 29334.339,E2 29334.339} C_VEL
LIN {X 0,Y 648.728,Z 333.411,A -85,B 0,C 180,E1 29331.58,E2 29331.58} C_VEL
LIN {X 0,Y 648.724,Z 333.424,A -85,B 0,C 180,E1 29328.351,E2 29328.351} C_VEL
LIN {X 0,Y 648.715,Z 333.395,A -85,B 0,C 180,E1 29325.54,E2 29325.54} C_VEL
LIN {X 0,Y 648.749,Z 333.415,A -85,B 0,C 180,E1 29322.417,E2 29322.417} C_VEL
LIN {X 0,Y 648.711,Z 333.415,A -85,B 0,C 180,E1 29319.52,E2 29319.52} C_VEL
LIN {X 0,Y 648.768,Z 333.394,A -85,B 0,C 180,E1 29316.473,E2 29316.473} C_VEL
LIN {X 0,Y 648.711,Z 333.418,A -85,B 0,C 180,E1 29313.548,E2 29313.548} C_VEL
LIN {X 0,Y 648.776,Z 333.417,A -85,B 0,C 180,E1 29310.545,E2 29310.545} C_VEL
LIN {X 0,Y 648.741,Z 333.509,A -85,B 0,C 180,E1 29307.772,E2 29307.772} C_VEL
LIN {X 0,Y 650.015,Z 336.904,A -85,B 0,C 180,E1 29307.321,E2 29307.321} C_VEL
LIN {X 0,Y 650.99,Z 338.597,A -85,B 0,C 180,E1 29307.062,E2 29307.062} C_VEL
LIN {X 0,Y 652.678,Z 341.829,A -85,B 0,C 180,E1 29306.634,E2 29306.634} C_VEL
LIN {X 0,Y 666.716,Z 361.533,A -85,B 0,C 180,E1 29304.916,E2 29304.916} C_VEL
LIN {X 0,Y 678.156,Z 378.707,A -85,B 0,C 180,E1 29303.594,E2 29303.594} C_VEL
LIN {X 0,Y 677.843,Z 396.468,A -85,B 0,C 180,E1 29303.354,E2 29303.354} C_VEL
LIN {X 0,Y 677.003,Z 404.176,A -85,B 0,C 180,E1 29303.312,E2 29303.312} C_VEL
LIN {X 0,Y 672.32,Z 424.863,A -85,B 0,C 180,E1 29303.417,E2 29303.417} C_VEL
LIN {X 0,Y 671.693,Z 431.47,A -85,B 0,C 180,E1 29303.373,E2 29303.373} C_VEL
LIN {X 0,Y 668.035,Z 644.675,A -85,B 0,C 180,E1 29300.519,E2 29300.519} C_VEL
LIN {X 0,Y 665.079,Z 819.772,A -85,B 0,C 180,E1 29298.216,E2 29298.216} C_VEL
LIN {X 0,Y 663.965,Z 847.543,A -85,B 0,C 180,E1 29297.694,E2 29297.694} C_VEL
LIN {X 0,Y 662.772,Z 870.899,A -85,B 0,C 180,E1 29297.113,E2 29297.113} C_VEL
LIN {X 0,Y 661.4,Z 894.362,A -85,B 0,C 180,E1 29296.395,E2 29296.395} C_VEL
LIN {X 0,Y 659.547,Z 921.554,A -85,B 0,C 180,E1 29295.377,E2 29295.377} C_VEL
LIN {X 0,Y 657.685,Z 945.601,A -85,B 0,C 180,E1 29294.306,E2 29294.306} C_VEL
LIN {X 0,Y 655.663,Z 970.049,A -85,B 0,C 180,E1 29293.039,E2 29293.039} C_VEL
LIN {X 0,Y 653.578,Z 993.934,A -85,B 0,C 180,E1 29291.601,E2 29291.601} C_VEL
LIN {X 0,Y 651.583,Z 1016.305,A -85,B 0,C 180,E1 29290.07,E2 29290.07} C_VEL
LIN {X 0,Y 649.54,Z 1038.499,A -85,B 0,C 180,E1 29288.342,E2 29288.342} C_VEL
LIN {X 0,Y 647.661,Z 1059.892,A -85,B 0,C 180,E1 29286.452,E2 29286.452} C_VEL
LIN {X 0,Y 645.862,Z 1080.427,A -85,B 0,C 180,E1 29284.394,E2 29284.394} C_VEL
LIN {X 0,Y 644.376,Z 1099.241,A -85,B 0,C 180,E1 29282.254,E2 29282.254} C_VEL
LIN {X 0,Y 643.082,Z 1116.717,A -85,B 0,C 180,E1 29279.997,E2 29279.997} C_VEL
LIN {X 0,Y 642.055,Z 1132.6,A -85,B 0,C 180,E1 29277.65,E2 29277.65} C_VEL
LIN {X 0,Y 641.255,Z 1146.655,A -85,B 0,C 180,E1 29275.26,E2 29275.26} C_VEL
LIN {X 0,Y 640.683,Z 1159.205,A -85,B 0,C 180,E1 29272.77,E2 29272.77} C_VEL
LIN {X 0,Y 640.319,Z 1169.304,A -85,B 0,C 180,E1 29270.378,E2 29270.378} C_VEL
LIN {X 0,Y 640.105,Z 1177.02,A -85,B 0,C 180,E1 29268.204,E2 29268.204} C_VEL
LIN {X 0,Y 639.996,Z 1183.534,A -85,B 0,C 180,E1 29265.96,E2 29265.96} C_VEL
LIN {X 0,Y 639.938,Z 1189.014,A -85,B 0,C 180,E1 29263.462,E2 29263.462} C_VEL
LIN {X 0,Y 639.915,Z 1192.46,A -85,B 0,C 180,E1 29261.172,E2 29261.172} C_VEL
LIN {X 0,Y 639.908,Z 1194.509,A -85,B 0,C 180,E1 29258.808,E2 29258.808} C_VEL
LIN {X 0,Y 639.908,Z 1194.867,A -85,B 0,C 180,E1 29256.389,E2 29256.389} C_VEL
LIN {X 0,Y 639.91,Z 1193.969,A -85,B 0,C 180,E1 29254.301,E2 29254.301} C_VEL
LIN {X 0,Y 639.924,Z 1191.482,A -85,B 0,C 180,E1 29251.97,E2 29251.97} C_VEL
LIN {X 0,Y 639.949,Z 1187.244,A -85,B 0,C 180,E1 29249.552,E2 29249.552} C_VEL
LIN {X 0,Y 640.025,Z 1181.814,A -85,B 0,C 180,E1 29247.314,E2 29247.314} C_VEL
LIN {X 0,Y 640.167,Z 1174.663,A -85,B 0,C 180,E1 29244.982,E2 29244.982} C_VEL
LIN {X 0,Y 640.471,Z 1165.001,A -85,B 0,C 180,E1 29242.46,E2 29242.46} C_VEL
LIN {X 0,Y 640.873,Z 1154.719,A -85,B 0,C 180,E1 29240.209,E2 29240.209} C_VEL
LIN {X 0,Y 641.504,Z 1142.196,A -85,B 0,C 180,E1 29237.854,E2 29237.854} C_VEL
LIN {X 0,Y 642.391,Z 1127.016,A -85,B 0,C 180,E1 29235.395,E2 29235.395} C_VEL
LIN {X 0,Y 643.57,Z 1110.06,A -85,B 0,C 180,E1 29233.018,E2 29233.018} C_VEL
LIN {X 0,Y 644.985,Z 1091.315,A -85,B 0,C 180,E1 29230.72,E2 29230.72} C_VEL
LIN {X 0,Y 646.619,Z 1071.571,A -85,B 0,C 180,E1 29228.597,E2 29228.597} C_VEL
LIN {X 0,Y 648.434,Z 1051.126,A -85,B 0,C 180,E1 29226.654,E2 29226.654} C_VEL
LIN {X 0,Y 650.433,Z 1028.941,A -85,B 0,C 180,E1 29224.798,E2 29224.798} C_VEL
LIN {X 0,Y 652.526,Z 1005.584,A -85,B 0,C 180,E1 29223.077,E2 29223.077} C_VEL
LIN {X 0,Y 654.68,Z 981.622,A -85,B 0,C 180,E1 29221.543,E2 29221.543} C_VEL
LIN {X 0,Y 656.678,Z 958.268,A -85,B 0,C 180,E1 29220.24,E2 29220.24} C_VEL
LIN {X 0,Y 658.62,Z 934.041,A -85,B 0,C 180,E1 29219.067,E2 29219.067} C_VEL
LIN {X 0,Y 660.386,Z 909.337,A -85,B 0,C 180,E1 29218.051,E2 29218.051} C_VEL
LIN {X 0,Y 661.916,Z 885.825,A -85,B 0,C 180,E1 29217.238,E2 29217.238} C_VEL
LIN {X 0,Y 663.466,Z 858.548,A -85,B 0,C 180,E1 29216.47,E2 29216.47} C_VEL
LIN {X 0,Y 664.556,Z 833.24,A -85,B 0,C 180,E1 29215.927,E2 29215.927} C_VEL
LIN {X 0,Y 665.398,Z 807.718,A -85,B 0,C 180,E1 29215.52,E2 29215.52} C_VEL
LIN {X 0,Y 668.988,Z 587.356,A -85,B 0,C 180,E1 29212.632,E2 29212.632} C_VEL
LIN {X 0,Y 672.581,Z 382.4,A -85,B 0,C 180,E1 29209.868,E2 29209.868} C_VEL
LIN {X 0,Y 658.7,Z 361.982,A -85,B 0,C 180,E1 29208.22,E2 29208.22} C_VEL
LIN {X 0,Y 648.424,Z 347.602,A -85,B 0,C 180,E1 29206.929,E2 29206.929} C_VEL
LIN {X 0,Y 643.526,Z 340.944,A -85,B 0,C 180,E1 29206.259,E2 29206.259} C_VEL
LIN {X 0,Y 642.297,Z 338.152,A -85,B 0,C 180,E1 29205.862,E2 29205.862} C_VEL
LIN {X 0,Y 640.79,Z 334.622,A -85,B 0,C 180,E1 29205.361,E2 29205.361} C_VEL
LIN {X 0,Y 640.728,Z 334.397,A -85,B 0,C 180,E1 29202.693,E2 29202.693} C_VEL
LIN {X 0,Y 640.796,Z 334.412,A -85,B 0,C 180,E1 29199.854,E2 29199.854} C_VEL
LIN {X 0,Y 640.738,Z 334.413,A -85,B 0,C 180,E1 29196.816,E2 29196.816} C_VEL
LIN {X 0,Y 640.742,Z 334.409,A -85,B 0,C 180,E1 29194.18,E2 29194.18} C_VEL
LIN {X 0,Y 640.777,Z 334.414,A -85,B 0,C 180,E1 29191.058,E2 29191.058} C_VEL
LIN {X 0,Y 640.732,Z 334.385,A -85,B 0,C 180,E1 29188.321,E2 29188.321} C_VEL
LIN {X 0,Y 640.81,Z 334.406,A -85,B 0,C 180,E1 29185.39,E2 29185.39} C_VEL
LIN {X 0,Y 640.736,Z 334.386,A -85,B 0,C 180,E1 29182.382,E2 29182.382} C_VEL
LIN {X 0,Y 640.747,Z 334.401,A -85,B 0,C 180,E1 29179.788,E2 29179.788} C_VEL
LIN {X 0,Y 640.775,Z 334.405,A -85,B 0,C 180,E1 29176.65,E2 29176.65} C_VEL
LIN {X 0,Y 640.737,Z 334.41,A -85,B 0,C 180,E1 29173.998,E2 29173.998} C_VEL
LIN {X 0,Y 640.778,Z 334.414,A -85,B 0,C 180,E1 29171.248,E2 29171.248} C_VEL
LIN {X 0,Y 640.752,Z 334.412,A -85,B 0,C 180,E1 29168.164,E2 29168.164} C_VEL
LIN {X 0,Y 640.74,Z 334.406,A -85,B 0,C 180,E1 29165.642,E2 29165.642} C_VEL
LIN {X 0,Y 640.821,Z 334.4,A -85,B 0,C 180,E1 29162.683,E2 29162.683} C_VEL
LIN {X 0,Y 640.742,Z 334.408,A -85,B 0,C 180,E1 29159.732,E2 29159.732} C_VEL
LIN {X 0,Y 640.765,Z 334.413,A -85,B 0,C 180,E1 29157.034,E2 29157.034} C_VEL
LIN {X 0,Y 640.759,Z 334.412,A -85,B 0,C 180,E1 29153.819,E2 29153.819} C_VEL
LIN {X 0,Y 640.746,Z 334.409,A -85,B 0,C 180,E1 29151.203,E2 29151.203} C_VEL
LIN {X 0,Y 640.821,Z 334.378,A -85,B 0,C 180,E1 29148.205,E2 29148.205} C_VEL
LIN {X 0,Y 640.744,Z 334.405,A -85,B 0,C 180,E1 29145.264,E2 29145.264} C_VEL
LIN {X 0,Y 640.778,Z 334.401,A -85,B 0,C 180,E1 29142.566,E2 29142.566} C_VEL
LIN {X 0,Y 640.761,Z 334.401,A -85,B 0,C 180,E1 29139.431,E2 29139.431} C_VEL
LIN {X 0,Y 640.749,Z 334.409,A -85,B 0,C 180,E1 29136.795,E2 29136.795} C_VEL
LIN {X 0,Y 640.822,Z 334.39,A -85,B 0,C 180,E1 29133.786,E2 29133.786} C_VEL
LIN {X 0,Y 640.749,Z 334.411,A -85,B 0,C 180,E1 29130.864,E2 29130.864} C_VEL
LIN {X 0,Y 640.792,Z 334.411,A -85,B 0,C 180,E1 29128.084,E2 29128.084} C_VEL
LIN {X 0,Y 640.76,Z 334.415,A -85,B 0,C 180,E1 29124.952,E2 29124.952} C_VEL
LIN {X 0,Y 640.758,Z 334.428,A -85,B 0,C 180,E1 29122.4,E2 29122.4} C_VEL
LIN {X 0,Y 642.118,Z 337.924,A -85,B 0,C 180,E1 29121.928,E2 29121.928} C_VEL
LIN {X 0,Y 643.151,Z 339.613,A -85,B 0,C 180,E1 29121.661,E2 29121.661} C_VEL
LIN {X 0,Y 648.593,Z 350.804,A -85,B 0,C 180,E1 29120.11,E2 29120.11} C_VEL
LIN {X 0,Y 662.821,Z 370.973,A -85,B 0,C 180,E1 29118.34,E2 29118.34} C_VEL
LIN {X 0,Y 672.703,Z 385.661,A -85,B 0,C 180,E1 29117.18,E2 29117.18} C_VEL
LIN {X 0,Y 669.034,Z 594.649,A -85,B 0,C 180,E1 29114.359,E2 29114.359} C_VEL
LIN {X 0,Y 665.394,Z 817.845,A -85,B 0,C 180,E1 29111.433,E2 29111.433} C_VEL
LIN {X 0,Y 664.546,Z 843.498,A -85,B 0,C 180,E1 29111.023,E2 29111.023} C_VEL
LIN {X 0,Y 663.523,Z 866.701,A -85,B 0,C 180,E1 29110.526,E2 29110.526} C_VEL
LIN {X 0,Y 662.132,Z 892.826,A -85,B 0,C 180,E1 29109.815,E2 29109.815} C_VEL
LIN {X 0,Y 660.419,Z 918.749,A -85,B 0,C 180,E1 29108.925,E2 29108.925} C_VEL
LIN {X 0,Y 658.811,Z 940.78,A -85,B 0,C 180,E1 29108.029,E2 29108.029} C_VEL
LIN {X 0,Y 657.097,Z 962.824,A -85,B 0,C 180,E1 29106.994,E2 29106.994} C_VEL
LIN {X 0,Y 654.914,Z 988.964,A -85,B 0,C 180,E1 29105.568,E2 29105.568} C_VEL
LIN {X 0,Y 652.993,Z 1010.386,A -85,B 0,C 180,E1 29104.221,E2 29104.221} C_VEL
LIN {X 0,Y 651.255,Z 1029.466,A -85,B 0,C 180,E1 29102.878,E2 29102.878} C_VEL
LIN {X 0,Y 649.322,Z 1051.291,A -85,B 0,C 180,E1 29101.157,E2 29101.157} C_VEL
LIN {X 0,Y 647.518,Z 1071.282,A -85,B 0,C 180,E1 29099.358,E2 29099.358} C_VEL
LIN {X 0,Y 646.097,Z 1087.697,A -85,B 0,C 180,E1 29097.721,E2 29097.721} C_VEL
LIN {X 0,Y 644.596,Z 1106.403,A -85,B 0,C 180,E1 29095.643,E2 29095.643} C_VEL
LIN {X 0,Y 643.325,Z 1122.989,A -85,B 0,C 180,E1 29093.542,E2 29093.542} C_VEL
LIN {X 0,Y 642.422,Z 1136.385,A -85,B 0,C 180,E1 29091.645,E2 29091.645} C_VEL
LIN {X 0,Y 641.561,Z 1151.1,A -85,B 0,C 180,E1 29089.293,E2 29089.293} C_VEL
LIN {X 0,Y 640.933,Z 1163.147,A -85,B 0,C 180,E1 29087.054,E2 29087.054} C_VEL
LIN {X 0,Y 640.55,Z 1172.31,A -85,B 0,C 180,E1 29085.11,E2 29085.11} C_VEL
LIN {X 0,Y 640.29,Z 1180.578,A -85,B 0,C 180,E1 29083.087,E2 29083.087} C_VEL
LIN {X 0,Y 640.073,Z 1188.479,A -85,B 0,C 180,E1 29080.804,E2 29080.804} C_VEL
LIN {X 0,Y 639.978,Z 1195.12,A -85,B 0,C 180,E1 29078.354,E2 29078.354} C_VEL
LIN {X 0,Y 639.931,Z 1199.724,A -85,B 0,C 180,E1 29076.099,E2 29076.099} C_VEL
LIN {X 0,Y 639.912,Z 1203.094,A -85,B 0,C 180,E1 29073.673,E2 29073.673} C_VEL
LIN {X 0,Y 639.914,Z 1204.669,A -85,B 0,C 180,E1 29071.343,E2 29071.343} C_VEL
LIN {X 0,Y 639.894,Z 1204.849,A -85,B 0,C 180,E1 29069.373,E2 29069.373} C_VEL
LIN {X 0,Y 639.91,Z 1203.941,A -85,B 0,C 180,E1 29067.313,E2 29067.313} C_VEL
LIN {X 0,Y 639.922,Z 1201.552,A -85,B 0,C 180,E1 29065.07,E2 29065.07} C_VEL
LIN {X 0,Y 639.953,Z 1197.347,A -85,B 0,C 180,E1 29062.639,E2 29062.639} C_VEL
LIN {X 0,Y 640.026,Z 1191.624,A -85,B 0,C 180,E1 29060.287,E2 29060.287} C_VEL
LIN {X 0,Y 640.164,Z 1184.591,A -85,B 0,C 180,E1 29058.011,E2 29058.011} C_VEL
LIN {X 0,Y 640.484,Z 1174.741,A -85,B 0,C 180,E1 29055.443,E2 29055.443} C_VEL
LIN {X 0,Y 640.843,Z 1165.001,A -85,B 0,C 180,E1 29053.317,E2 29053.317} C_VEL
LIN {X 0,Y 641.35,Z 1154.761,A -85,B 0,C 180,E1 29051.362,E2 29051.362} C_VEL
LIN {X 0,Y 642.053,Z 1142.531,A -85,B 0,C 180,E1 29049.298,E2 29049.298} C_VEL
LIN {X 0,Y 643.082,Z 1126.501,A -85,B 0,C 180,E1 29046.933,E2 29046.933} C_VEL
LIN {X 0,Y 644.144,Z 1111.858,A -85,B 0,C 180,E1 29045.026,E2 29045.026} C_VEL
LIN {X 0,Y 645.467,Z 1095.435,A -85,B 0,C 180,E1 29043.107,E2 29043.107} C_VEL
LIN {X 0,Y 647.156,Z 1075.337,A -85,B 0,C 180,E1 29041.03,E2 29041.03} C_VEL
LIN {X 0,Y 648.61,Z 1058.942,A -85,B 0,C 180,E1 29039.514,E2 29039.514} C_VEL
LIN {X 0,Y 650.17,Z 1041.626,A -85,B 0,C 180,E1 29038.061,E2 29038.061} C_VEL
LIN {X 0,Y 652.2,Z 1019.55,A -85,B 0,C 180,E1 29036.397,E2 29036.397} C_VEL
LIN {X 0,Y 654.232,Z 996.179,A -85,B 0,C 180,E1 29034.867,E2 29034.867} C_VEL
LIN {X 0,Y 655.998,Z 975.858,A -85,B 0,C 180,E1 29033.691,E2 29033.691} C_VEL
LIN {X 0,Y 657.988,Z 952.264,A -85,B 0,C 180,E1 29032.49,E2 29032.49} C_VEL
LIN {X 0,Y 659.917,Z 926.451,A -85,B 0,C 180,E1 29031.374,E2 29031.374} C_VEL
LIN {X 0,Y 661.328,Z 904.877,A -85,B 0,C 180,E1 29030.58,E2 29030.58} C_VEL
LIN {X 0,Y 662.652,Z 883.013,A -85,B 0,C 180,E1 29029.901,E2 29029.901} C_VEL
LIN {X 0,Y 663.947,Z 858.262,A -85,B 0,C 180,E1 29029.275,E2 29029.275} C_VEL
LIN {X 0,Y 665.053,Z 829.748,A -85,B 0,C 180,E1 29028.74,E2 29028.74} C_VEL
LIN {X 0,Y 666.538,Z 746.82,A -85,B 0,C 180,E1 29027.643,E2 29027.643} C_VEL
LIN {X 0,Y 670.249,Z 524.283,A -85,B 0,C 180,E1 29024.702,E2 29024.702} C_VEL
LIN {X 0,Y 672.614,Z 385.439,A -85,B 0,C 180,E1 29022.809,E2 29022.809} C_VEL
LIN {X 0,Y 656.333,Z 361.641,A -85,B 0,C 180,E1 29020.869,E2 29020.869} C_VEL
LIN {X 0,Y 648.027,Z 349.886,A -85,B 0,C 180,E1 29019.792,E2 29019.792} C_VEL
LIN {X 0,Y 644.166,Z 342.04,A -85,B 0,C 180,E1 29018.672,E2 29018.672} C_VEL
LIN {X 0,Y 642.542,Z 338.464,A -85,B 0,C 180,E1 29018.155,E2 29018.155} C_VEL
LIN {X 0,Y 640.99,Z 335.544,A -85,B 0,C 180,E1 29017.697,E2 29017.697} C_VEL
LIN {X 0,Y 640.759,Z 334.417,A -85,B 0,C 180,E1 29017.525,E2 29017.525} C_VEL
LIN {X 0,Y 640.797,Z 334.41,A -85,B 0,C 180,E1 29014.685,E2 29014.685} C_VEL
LIN {X 0,Y 640.764,Z 334.385,A -85,B 0,C 180,E1 29011.518,E2 29011.518} C_VEL
LIN {X 0,Y 640.769,Z 334.411,A -85,B 0,C 180,E1 29008.828,E2 29008.828} C_VEL
LIN {X 0,Y 640.803,Z 334.397,A -85,B 0,C 180,E1 29005.708,E2 29005.708} C_VEL
LIN {X 0,Y 640.758,Z 334.388,A -85,B 0,C 180,E1 29002.865,E2 29002.865} C_VEL
LIN {X 0,Y 640.837,Z 334.409,A -85,B 0,C 180,E1 28999.81,E2 28999.81} C_VEL
LIN {X 0,Y 640.76,Z 334.391,A -85,B 0,C 180,E1 28996.78,E2 28996.78} C_VEL
LIN {X 0,Y 640.832,Z 334.399,A -85,B 0,C 180,E1 28993.811,E2 28993.811} C_VEL
LIN {X 0,Y 640.766,Z 334.404,A -85,B 0,C 180,E1 28990.793,E2 28990.793} C_VEL
LIN {X 0,Y 640.793,Z 334.398,A -85,B 0,C 180,E1 28987.983,E2 28987.983} C_VEL
LIN {X 0,Y 640.781,Z 334.41,A -85,B 0,C 180,E1 28984.834,E2 28984.834} C_VEL
LIN {X 0,Y 640.772,Z 334.392,A -85,B 0,C 180,E1 28982.057,E2 28982.057} C_VEL
LIN {X 0,Y 640.811,Z 334.41,A -85,B 0,C 180,E1 28978.927,E2 28978.927} C_VEL
LIN {X 0,Y 640.764,Z 334.382,A -85,B 0,C 180,E1 28976.063,E2 28976.063} C_VEL
LIN {X 0,Y 640.838,Z 334.408,A -85,B 0,C 180,E1 28973.01,E2 28973.01} C_VEL
LIN {X 0,Y 640.765,Z 334.386,A -85,B 0,C 180,E1 28970.025,E2 28970.025} C_VEL
LIN {X 0,Y 640.833,Z 334.4,A -85,B 0,C 180,E1 28967.016,E2 28967.016} C_VEL
LIN {X 0,Y 640.771,Z 334.405,A -85,B 0,C 180,E1 28963.966,E2 28963.966} C_VEL
LIN {X 0,Y 640.814,Z 334.384,A -85,B 0,C 180,E1 28961.061,E2 28961.061} C_VEL
LIN {X 0,Y 640.779,Z 334.408,A -85,B 0,C 180,E1 28957.951,E2 28957.951} C_VEL
LIN {X 0,Y 640.794,Z 334.4,A -85,B 0,C 180,E1 28955.083,E2 28955.083} C_VEL
LIN {X 0,Y 640.787,Z 334.413,A -85,B 0,C 180,E1 28951.836,E2 28951.836} C_VEL
LIN {X 0,Y 640.796,Z 334.405,A -85,B 0,C 180,E1 28948.94,E2 28948.94} C_VEL
LIN {X 0,Y 640.835,Z 334.426,A -85,B 0,C 180,E1 28948.589,E2 28948.589} C_VEL
LIN {X 0,Y 642.027,Z 337.727,A -85,B 0,C 180,E1 28948.132,E2 28948.132} C_VEL
LIN {X 0,Y 643.002,Z 339.303,A -85,B 0,C 180,E1 28947.871,E2 28947.871} C_VEL
LIN {X 0,Y 644.133,Z 341.926,A -85,B 0,C 180,E1 28947.54,E2 28947.54} C_VEL
LIN {X 0,Y 650.484,Z 350.469,A -85,B 0,C 180,E1 28946.718,E2 28946.718} C_VEL
LIN {X 0,Y 662.593,Z 367.42,A -85,B 0,C 180,E1 28945.22,E2 28945.22} C_VEL
LIN {X 0,Y 672.584,Z 382.555,A -85,B 0,C 180,E1 28944.04,E2 28944.04} C_VEL
LIN {X 0,Y 671.693,Z 431.47,A -85,B 0,C 180,E1 28943.373,E2 28943.373} C_VEL
LIN {X 0,Y 670.874,Z 439.176,A -85,B 0,C 180,E1 28943.329,E2 28943.329} C_VEL
LIN {X 0,Y 666.172,Z 459.863,A -85,B 0,C 180,E1 28943.437,E2 28943.437} C_VEL
LIN {X 0,Y 665.528,Z 466.474,A -85,B 0,C 180,E1 28943.394,E2 28943.394} C_VEL
LIN {X 0,Y 661.483,Z 687.196,A -85,B 0,C 180,E1 28940.435,E2 28940.435} C_VEL
LIN {X 0,Y 659.051,Z 820.07,A -85,B 0,C 180,E1 28938.673,E2 28938.673} C_VEL
LIN {X 0,Y 657.871,Z 847.635,A -85,B 0,C 180,E1 28938.15,E2 28938.15} C_VEL
LIN {X 0,Y 656.609,Z 870.8,A -85,B 0,C 180,E1 28937.571,E2 28937.571} C_VEL
LIN {X 0,Y 655.136,Z 894.404,A -85,B 0,C 180,E1 28936.846,E2 28936.846} C_VEL
LIN {X 0,Y 653.166,Z 921.442,A -85,B 0,C 180,E1 28935.828,E2 28935.828} C_VEL
LIN {X 0,Y 651.179,Z 945.489,A -85,B 0,C 180,E1 28934.749,E2 28934.749} C_VEL
LIN {X 0,Y 649.005,Z 969.916,A -85,B 0,C 180,E1 28933.477,E2 28933.477} C_VEL
LIN {X 0,Y 646.74,Z 993.911,A -85,B 0,C 180,E1 28932.022,E2 28932.022} C_VEL
LIN {X 0,Y 644.609,Z 1016.295,A -85,B 0,C 180,E1 28930.477,E2 28930.477} C_VEL
LIN {X 0,Y 642.336,Z 1039.094,A -85,B 0,C 180,E1 28928.68,E2 28928.68} C_VEL
LIN {X 0,Y 640.307,Z 1060.49,A -85,B 0,C 180,E1 28926.765,E2 28926.765} C_VEL
LIN {X 0,Y 638.369,Z 1080.967,A -85,B 0,C 180,E1 28924.682,E2 28924.682} C_VEL
LIN {X 0,Y 636.806,Z 1099.178,A -85,B 0,C 180,E1 28922.585,E2 28922.585} C_VEL
LIN {X 0,Y 635.414,Z 1116.389,A -85,B 0,C 180,E1 28920.339,E2 28920.339} C_VEL
LIN {X 0,Y 634.269,Z 1132.599,A -85,B 0,C 180,E1 28917.917,E2 28917.917} C_VEL
LIN {X 0,Y 633.405,Z 1146.481,A -85,B 0,C 180,E1 28915.527,E2 28915.527} C_VEL
LIN {X 0,Y 632.775,Z 1159.21,A -85,B 0,C 180,E1 28912.972,E2 28912.972} C_VEL
LIN {X 0,Y 632.358,Z 1169.31,A -85,B 0,C 180,E1 28910.549,E2 28910.549} C_VEL
LIN {X 0,Y 632.132,Z 1177.022,A -85,B 0,C 180,E1 28908.346,E2 28908.346} C_VEL
LIN {X 0,Y 632.002,Z 1183.788,A -85,B 0,C 180,E1 28905.978,E2 28905.978} C_VEL
LIN {X 0,Y 631.939,Z 1189.174,A -85,B 0,C 180,E1 28903.449,E2 28903.449} C_VEL
LIN {X 0,Y 631.917,Z 1192.518,A -85,B 0,C 180,E1 28901.175,E2 28901.175} C_VEL
LIN {X 0,Y 631.907,Z 1194.564,A -85,B 0,C 180,E1 28898.737,E2 28898.737} C_VEL
LIN {X 0,Y 631.91,Z 1194.861,A -85,B 0,C 180,E1 28896.359,E2 28896.359} C_VEL
LIN {X 0,Y 631.91,Z 1193.964,A -85,B 0,C 180,E1 28894.265,E2 28894.265} C_VEL
LIN {X 0,Y 631.923,Z 1191.479,A -85,B 0,C 180,E1 28891.904,E2 28891.904} C_VEL
LIN {X 0,Y 631.952,Z 1187.239,A -85,B 0,C 180,E1 28889.456,E2 28889.456} C_VEL
LIN {X 0,Y 632.035,Z 1181.807,A -85,B 0,C 180,E1 28887.189,E2 28887.189} C_VEL
LIN {X 0,Y 632.197,Z 1174.66,A -85,B 0,C 180,E1 28884.828,E2 28884.828} C_VEL
LIN {X 0,Y 632.526,Z 1165.016,A -85,B 0,C 180,E1 28882.278,E2 28882.278} C_VEL
LIN {X 0,Y 632.968,Z 1154.723,A -85,B 0,C 180,E1 28879.994,E2 28879.994} C_VEL
LIN {X 0,Y 633.658,Z 1142.202,A -85,B 0,C 180,E1 28877.608,E2 28877.608} C_VEL
LIN {X 0,Y 634.626,Z 1127.02,A -85,B 0,C 180,E1 28875.119,E2 28875.119} C_VEL
LIN {X 0,Y 635.913,Z 1110.067,A -85,B 0,C 180,E1 28872.712,E2 28872.712} C_VEL
LIN {X 0,Y 637.476,Z 1091.332,A -85,B 0,C 180,E1 28870.388,E2 28870.388} C_VEL
LIN {X 0,Y 639.223,Z 1071.584,A -85,B 0,C 180,E1 28868.241,E2 28868.241} C_VEL
LIN {X 0,Y 641.23,Z 1050.874,A -85,B 0,C 180,E1 28866.253,E2 28866.253} C_VEL
LIN {X 0,Y 643.353,Z 1028.953,A -85,B 0,C 180,E1 28864.402,E2 28864.402} C_VEL
LIN {X 0,Y 645.623,Z 1005.592,A -85,B 0,C 180,E1 28862.666,E2 28862.666} C_VEL
LIN {X 0,Y 647.936,Z 981.622,A -85,B 0,C 180,E1 28861.118,E2 28861.118} C_VEL
LIN {X 0,Y 649.993,Z 959.141,A -85,B 0,C 180,E1 28859.852,E2 28859.852} C_VEL
LIN {X 0,Y 652.092,Z 934.846,A -85,B 0,C 180,E1 28858.659,E2 28858.659} C_VEL
LIN {X 0,Y 654.045,Z 909.302,A -85,B 0,C 180,E1 28857.601,E2 28857.601} C_VEL
LIN {X 0,Y 655.637,Z 886.49,A -85,B 0,C 180,E1 28856.806,E2 28856.806} C_VEL
LIN {X 0,Y 657.28,Z 859.821,A -85,B 0,C 180,E1 28856.043,E2 28856.043} C_VEL
LIN {X 0,Y 658.477,Z 833.879,A -85,B 0,C 180,E1 28855.479,E2 28855.479} C_VEL
LIN {X 0,Y 659.35,Z 809.256,A -85,B 0,C 180,E1 28855.08,E2 28855.08} C_VEL
LIN {X 0,Y 663.223,Z 589.519,A -85,B 0,C 180,E1 28852.175,E2 28852.175} C_VEL
LIN {X 0,Y 667.059,Z 386.213,A -85,B 0,C 180,E1 28849.414,E2 28849.414} C_VEL
LIN {X 0,Y 654.431,Z 367.608,A -85,B 0,C 180,E1 28847.884,E2 28847.884} C_VEL
LIN {X 0,Y 644.159,Z 353.266,A -85,B 0,C 180,E1 28846.57,E2 28846.57} C_VEL
LIN {X 0,Y 635.297,Z 341.054,A -85,B 0,C 180,E1 28845.349,E2 28845.349} C_VEL
LIN {X 0,Y 633.924,Z 338.621,A -85,B 0,C 180,E1 28844.962,E2 28844.962} C_VEL
LIN {X 0,Y 632.799,Z 335.409,A -85,B 0,C 180,E1 28844.496,E2 28844.496} C_VEL
LIN {X 0,Y 632.837,Z 335.383,A -85,B 0,C 180,E1 28841.368,E2 28841.368} C_VEL
LIN {X 0,Y 632.791,Z 335.406,A -85,B 0,C 180,E1 28838.62,E2 28838.62} C_VEL
LIN {X 0,Y 632.853,Z 335.404,A -85,B 0,C 180,E1 28835.774,E2 28835.774} C_VEL
LIN {X 0,Y 632.8,Z 335.402,A -85,B 0,C 180,E1 28832.711,E2 28832.711} C_VEL
LIN {X 0,Y 632.808,Z 335.405,A -85,B 0,C 180,E1 28830.059,E2 28830.059} C_VEL
LIN {X 0,Y 632.825,Z 335.375,A -85,B 0,C 180,E1 28826.865,E2 28826.865} C_VEL
LIN {X 0,Y 632.797,Z 335.403,A -85,B 0,C 180,E1 28824.158,E2 28824.158} C_VEL
LIN {X 0,Y 632.878,Z 335.358,A -85,B 0,C 180,E1 28821.211,E2 28821.211} C_VEL
LIN {X 0,Y 632.801,Z 335.402,A -85,B 0,C 180,E1 28818.232,E2 28818.232} C_VEL
LIN {X 0,Y 632.824,Z 335.399,A -85,B 0,C 180,E1 28815.488,E2 28815.488} C_VEL
LIN {X 0,Y 632.816,Z 335.401,A -85,B 0,C 180,E1 28812.316,E2 28812.316} C_VEL
LIN {X 0,Y 632.804,Z 335.393,A -85,B 0,C 180,E1 28809.618,E2 28809.618} C_VEL
LIN {X 0,Y 632.859,Z 335.389,A -85,B 0,C 180,E1 28806.532,E2 28806.532} C_VEL
LIN {X 0,Y 632.802,Z 335.401,A -85,B 0,C 180,E1 28803.714,E2 28803.714} C_VEL
LIN {X 0,Y 632.866,Z 335.401,A -85,B 0,C 180,E1 28800.815,E2 28800.815} C_VEL
LIN {X 0,Y 632.807,Z 335.401,A -85,B 0,C 180,E1 28797.736,E2 28797.736} C_VEL
LIN {X 0,Y 632.823,Z 335.392,A -85,B 0,C 180,E1 28795.015,E2 28795.015} C_VEL
LIN {X 0,Y 632.825,Z 335.396,A -85,B 0,C 180,E1 28791.825,E2 28791.825} C_VEL
LIN {X 0,Y 632.806,Z 335.399,A -85,B 0,C 180,E1 28789.162,E2 28789.162} C_VEL
LIN {X 0,Y 632.881,Z 335.364,A -85,B 0,C 180,E1 28786.105,E2 28786.105} C_VEL
LIN {X 0,Y 632.808,Z 335.401,A -85,B 0,C 180,E1 28783.193,E2 28783.193} C_VEL
LIN {X 0,Y 632.871,Z 335.361,A -85,B 0,C 180,E1 28780.238,E2 28780.238} C_VEL
LIN {X 0,Y 632.814,Z 335.398,A -85,B 0,C 180,E1 28777.225,E2 28777.225} C_VEL
LIN {X 0,Y 632.819,Z 335.368,A -85,B 0,C 180,E1 28774.547,E2 28774.547} C_VEL
LIN {X 0,Y 632.832,Z 335.395,A -85,B 0,C 180,E1 28771.293,E2 28771.293} C_VEL
LIN {X 0,Y 632.812,Z 335.398,A -85,B 0,C 180,E1 28768.678,E2 28768.678} C_VEL
LIN {X 0,Y 632.888,Z 335.397,A -85,B 0,C 180,E1 28765.666,E2 28765.666} C_VEL
LIN {X 0,Y 632.878,Z 335.632,A -85,B 0,C 180,E1 28763.178,E2 28763.178} C_VEL
LIN {X 0,Y 634.111,Z 338.875,A -85,B 0,C 180,E1 28762.735,E2 28762.735} C_VEL
LIN {X 0,Y 635.128,Z 340.557,A -85,B 0,C 180,E1 28762.464,E2 28762.464} C_VEL
LIN {X 0,Y 639.818,Z 350.245,A -85,B 0,C 180,E1 28761.065,E2 28761.065} C_VEL
LIN {X 0,Y 650.214,Z 364.769,A -85,B 0,C 180,E1 28759.705,E2 28759.705} C_VEL
LIN {X 0,Y 662.44,Z 382.394,A -85,B 0,C 180,E1 28758.195,E2 28758.195} C_VEL
LIN {X 0,Y 667.17,Z 389.67,A -85,B 0,C 180,E1 28757.63,E2 28757.63} C_VEL
LIN {X 0,Y 663.27,Z 596.939,A -85,B 0,C 180,E1 28754.814,E2 28754.814} C_VEL
LIN {X 0,Y 659.342,Z 819.427,A -85,B 0,C 180,E1 28751.872,E2 28751.872} C_VEL
LIN {X 0,Y 658.473,Z 843.96,A -85,B 0,C 180,E1 28751.474,E2 28751.474} C_VEL
LIN {X 0,Y 657.397,Z 866.811,A -85,B 0,C 180,E1 28750.981,E2 28750.981} C_VEL
LIN {X 0,Y 655.94,Z 892.517,A -85,B 0,C 180,E1 28750.278,E2 28750.278} C_VEL
LIN {X 0,Y 654.083,Z 918.746,A -85,B 0,C 180,E1 28749.374,E2 28749.374} C_VEL
LIN {X 0,Y 652.374,Z 940.609,A -85,B 0,C 180,E1 28748.481,E2 28748.481} C_VEL
LIN {X 0,Y 650.527,Z 962.727,A -85,B 0,C 180,E1 28747.436,E2 28747.436} C_VEL
LIN {X 0,Y 648.184,Z 988.961,A -85,B 0,C 180,E1 28745.995,E2 28745.995} C_VEL
LIN {X 0,Y 646.229,Z 1009.336,A -85,B 0,C 180,E1 28744.707,E2 28744.707} C_VEL
LIN {X 0,Y 644.436,Z 1027.718,A -85,B 0,C 180,E1 28743.41,E2 28743.41} C_VEL
LIN {X 0,Y 642.595,Z 1046.485,A -85,B 0,C 180,E1 28741.94,E2 28741.94} C_VEL
LIN {X 0,Y 640.404,Z 1069.081,A -85,B 0,C 180,E1 28739.94,E2 28739.94} C_VEL
LIN {X 0,Y 638.845,Z 1085.923,A -85,B 0,C 180,E1 28738.258,E2 28738.258} C_VEL
LIN {X 0,Y 637.368,Z 1102.229,A -85,B 0,C 180,E1 28736.456,E2 28736.456} C_VEL
LIN {X 0,Y 635.893,Z 1120.245,A -85,B 0,C 180,E1 28734.216,E2 28734.216} C_VEL
LIN {X 0,Y 634.769,Z 1134.906,A -85,B 0,C 180,E1 28732.146,E2 28732.146} C_VEL
LIN {X 0,Y 633.906,Z 1147.733,A -85,B 0,C 180,E1 28730.112,E2 28730.112} C_VEL
LIN {X 0,Y 633.149,Z 1161.287,A -85,B 0,C 180,E1 28727.65,E2 28727.65} C_VEL
LIN {X 0,Y 632.659,Z 1171.079,A -85,B 0,C 180,E1 28725.585,E2 28725.585} C_VEL
LIN {X 0,Y 632.373,Z 1179.16,A -85,B 0,C 180,E1 28723.626,E2 28723.626} C_VEL
LIN {X 0,Y 632.15,Z 1186.71,A -85,B 0,C 180,E1 28721.495,E2 28721.495} C_VEL
LIN {X 0,Y 632.004,Z 1193.595,A -85,B 0,C 180,E1 28719.103,E2 28719.103} C_VEL
LIN {X 0,Y 631.938,Z 1198.922,A -85,B 0,C 180,E1 28716.632,E2 28716.632} C_VEL
LIN {X 0,Y 631.917,Z 1202.357,A -85,B 0,C 180,E1 28714.356,E2 28714.356} C_VEL
LIN {X 0,Y 631.911,Z 1204.438,A -85,B 0,C 180,E1 28711.995,E2 28711.995} C_VEL
LIN {X 0,Y 631.892,Z 1204.894,A -85,B 0,C 180,E1 28709.547,E2 28709.547} C_VEL
LIN {X 0,Y 631.908,Z 1204.007,A -85,B 0,C 180,E1 28707.37,E2 28707.37} C_VEL
LIN {X 0,Y 631.921,Z 1201.674,A -85,B 0,C 180,E1 28705.099,E2 28705.099} C_VEL
LIN {X 0,Y 631.956,Z 1197.542,A -85,B 0,C 180,E1 28702.637,E2 28702.637} C_VEL
LIN {X 0,Y 632.034,Z 1191.875,A -85,B 0,C 180,E1 28700.255,E2 28700.255} C_VEL
LIN {X 0,Y 632.182,Z 1184.891,A -85,B 0,C 180,E1 28697.95,E2 28697.95} C_VEL
LIN {X 0,Y 632.529,Z 1175.145,A -85,B 0,C 180,E1 28695.35,E2 28695.35} C_VEL
LIN {X 0,Y 632.943,Z 1165,A -85,B 0,C 180,E1 28693.102,E2 28693.102} C_VEL
LIN {X 0,Y 633.497,Z 1154.763,A -85,B 0,C 180,E1 28691.122,E2 28691.122} C_VEL
LIN {X 0,Y 634.299,Z 1141.95,A -85,B 0,C 180,E1 28688.937,E2 28688.937} C_VEL
LIN {X 0,Y 635.434,Z 1125.798,A -85,B 0,C 180,E1 28686.541,E2 28686.541} C_VEL
LIN {X 0,Y 636.629,Z 1111.083,A -85,B 0,C 180,E1 28684.611,E2 28684.611} C_VEL
LIN {X 0,Y 638.206,Z 1092.836,A -85,B 0,C 180,E1 28682.47,E2 28682.47} C_VEL
LIN {X 0,Y 639.969,Z 1073.816,A -85,B 0,C 180,E1 28680.519,E2 28680.519} C_VEL
LIN {X 0,Y 641.533,Z 1057.513,A -85,B 0,C 180,E1 28679.007,E2 28679.007} C_VEL
LIN {X 0,Y 643.319,Z 1039.19,A -85,B 0,C 180,E1 28677.469,E2 28677.469} C_VEL
LIN {X 0,Y 645.642,Z 1015.192,A -85,B 0,C 180,E1 28675.688,E2 28675.688} C_VEL
LIN {X 0,Y 647.617,Z 994.635,A -85,B 0,C 180,E1 28674.351,E2 28674.351} C_VEL
LIN {X 0,Y 649.503,Z 974.415,A -85,B 0,C 180,E1 28673.181,E2 28673.181} C_VEL
LIN {X 0,Y 651.753,Z 949.295,A -85,B 0,C 180,E1 28671.908,E2 28671.908} C_VEL
LIN {X 0,Y 653.674,Z 924.585,A -85,B 0,C 180,E1 28670.854,E2 28670.854} C_VEL
LIN {X 0,Y 655.115,Z 904.134,A -85,B 0,C 180,E1 28670.104,E2 28670.104} C_VEL
LIN {X 0,Y 656.512,Z 882.385,A -85,B 0,C 180,E1 28669.428,E2 28669.428} C_VEL
LIN {X 0,Y 657.909,Z 857.374,A -85,B 0,C 180,E1 28668.797,E2 28668.797} C_VEL
LIN {X 0,Y 659.042,Z 829.291,A -85,B 0,C 180,E1 28668.273,E2 28668.273} C_VEL
LIN {X 0,Y 660.722,Z 741.103,A -85,B 0,C 180,E1 28667.099,E2 28667.099} C_VEL
LIN {X 0,Y 664.731,Z 518.504,A -85,B 0,C 180,E1 28664.131,E2 28664.131} C_VEL
LIN {X 0,Y 667.125,Z 389.323,A -85,B 0,C 180,E1 28662.36,E2 28662.36} C_VEL
LIN {X 0,Y 652.194,Z 367.5,A -85,B 0,C 180,E1 28660.545,E2 28660.545} C_VEL
LIN {X 0,Y 641.851,Z 353.05,A -85,B 0,C 180,E1 28659.205,E2 28659.205} C_VEL
LIN {X 0,Y 639.655,Z 349.818,A -85,B 0,C 180,E1 28658.883,E2 28658.883} C_VEL
LIN {X 0,Y 636.777,Z 343.833,A -85,B 0,C 180,E1 28657.991,E2 28657.991} C_VEL
LIN {X 0,Y 634.706,Z 339.65,A -85,B 0,C 180,E1 28657.338,E2 28657.338} C_VEL
LIN {X 0,Y 633.004,Z 336.251,A -85,B 0,C 180,E1 28656.791,E2 28656.791} C_VEL
LIN {X 0,Y 632.865,Z 335.401,A -85,B 0,C 180,E1 28656.671,E2 28656.671} C_VEL
LIN {X 0,Y 632.828,Z 335.402,A -85,B 0,C 180,E1 28653.574,E2 28653.574} C_VEL
LIN {X 0,Y 632.833,Z 335.374,A -85,B 0,C 180,E1 28650.792,E2 28650.792} C_VEL
LIN {X 0,Y 632.84,Z 335.372,A -85,B 0,C 180,E1 28647.577,E2 28647.577} C_VEL
LIN {X 0,Y 632.828,Z 335.401,A -85,B 0,C 180,E1 28644.753,E2 28644.753} C_VEL
LIN {X 0,Y 632.865,Z 335.373,A -85,B 0,C 180,E1 28641.6,E2 28641.6} C_VEL
LIN {X 0,Y 632.823,Z 335.392,A -85,B 0,C 180,E1 28638.804,E2 28638.804} C_VEL
LIN {X 0,Y 632.895,Z 335.383,A -85,B 0,C 180,E1 28635.768,E2 28635.768} C_VEL
LIN {X 0,Y 632.822,Z 335.374,A -85,B 0,C 180,E1 28632.78,E2 28632.78} C_VEL
LIN {X 0,Y 632.869,Z 335.393,A -85,B 0,C 180,E1 28629.917,E2 28629.917} C_VEL
LIN {X 0,Y 632.832,Z 335.369,A -85,B 0,C 180,E1 28626.806,E2 28626.806} C_VEL
LIN {X 0,Y 632.844,Z 335.398,A -85,B 0,C 180,E1 28623.986,E2 28623.986} C_VEL
LIN {X 0,Y 632.84,Z 335.373,A -85,B 0,C 180,E1 28620.724,E2 28620.724} C_VEL
LIN {X 0,Y 632.838,Z 335.398,A -85,B 0,C 180,E1 28617.917,E2 28617.917} C_VEL
LIN {X 0,Y 632.861,Z 335.375,A -85,B 0,C 180,E1 28614.742,E2 28614.742} C_VEL
LIN {X 0,Y 632.83,Z 335.392,A -85,B 0,C 180,E1 28611.916,E2 28611.916} C_VEL
LIN {X 0,Y 632.887,Z 335.385,A -85,B 0,C 180,E1 28608.795,E2 28608.795} C_VEL
LIN {X 0,Y 632.828,Z 335.372,A -85,B 0,C 180,E1 28605.824,E2 28605.824} C_VEL
LIN {X 0,Y 632.897,Z 335.396,A -85,B 0,C 180,E1 28602.816,E2 28602.816} C_VEL
LIN {X 0,Y 632.83,Z 335.383,A -85,B 0,C 180,E1 28599.755,E2 28599.755} C_VEL
LIN {X 0,Y 632.889,Z 335.372,A -85,B 0,C 180,E1 28596.834,E2 28596.834} C_VEL
LIN {X 0,Y 632.839,Z 335.397,A -85,B 0,C 180,E1 28593.743,E2 28593.743} C_VEL
LIN {X 0,Y 632.88,Z 335.396,A -85,B 0,C 180,E1 28590.778,E2 28590.778} C_VEL
LIN {X 0,Y 632.844,Z 335.458,A -85,B 0,C 180,E1 28589.461,E2 28589.461} C_VEL
LIN {X 0,Y 634.131,Z 338.832,A -85,B 0,C 180,E1 28588.962,E2 28588.962} C_VEL
LIN {X 0,Y 635.16,Z 340.201,A -85,B 0,C 180,E1 28588.701,E2 28588.701} C_VEL
LIN {X 0,Y 635.992,Z 342.228,A -85,B 0,C 180,E1 28588.457,E2 28588.457} C_VEL
LIN {X 0,Y 646.684,Z 356.67,A -85,B 0,C 180,E1 28587.013,E2 28587.013} C_VEL
LIN {X 0,Y 658.632,Z 373.54,A -85,B 0,C 180,E1 28585.51,E2 28585.51} C_VEL
LIN {X 0,Y 667.058,Z 386.347,A -85,B 0,C 180,E1 28584.494,E2 28584.494} C_VEL
LIN {X 0,Y 665.528,Z 466.474,A -85,B 0,C 180,E1 28583.394,E2 28583.394} C_VEL
LIN {X 0,Y 664.69,Z 474.179,A -85,B 0,C 180,E1 28583.352,E2 28583.352} C_VEL
LIN {X 0,Y 659.942,Z 494.855,A -85,B 0,C 180,E1 28583.465,E2 28583.465} C_VEL
LIN {X 0,Y 659.29,Z 501.464,A -85,B 0,C 180,E1 28583.422,E2 28583.422} C_VEL
LIN {X 0,Y 655.105,Z 717.746,A -85,B 0,C 180,E1 28580.512,E2 28580.512} C_VEL
LIN {X 0,Y 653.061,Z 820.487,A -85,B 0,C 180,E1 28579.135,E2 28579.135} C_VEL
LIN {X 0,Y 651.819,Z 847.728,A -85,B 0,C 180,E1 28578.614,E2 28578.614} C_VEL
LIN {X 0,Y 650.501,Z 870.518,A -85,B 0,C 180,E1 28578.043,E2 28578.043} C_VEL
LIN {X 0,Y 648.962,Z 893.698,A -85,B 0,C 180,E1 28577.329,E2 28577.329} C_VEL
LIN {X 0,Y 646.919,Z 920.321,A -85,B 0,C 180,E1 28576.33,E2 28576.33} C_VEL
LIN {X 0,Y 644.907,Z 943.245,A -85,B 0,C 180,E1 28575.304,E2 28575.304} C_VEL
LIN {X 0,Y 642.846,Z 965.3,A -85,B 0,C 180,E1 28574.171,E2 28574.171} C_VEL
LIN {X 0,Y 640.245,Z 990.953,A -85,B 0,C 180,E1 28572.644,E2 28572.644} C_VEL
LIN {X 0,Y 637.876,Z 1014.068,A -85,B 0,C 180,E1 28571.054,E2 28571.054} C_VEL
LIN {X 0,Y 635.369,Z 1037.832,A -85,B 0,C 180,E1 28569.185,E2 28569.185} C_VEL
LIN {X 0,Y 633.092,Z 1059.704,A -85,B 0,C 180,E1 28567.22,E2 28567.22} C_VEL
LIN {X 0,Y 631.032,Z 1080.285,A -85,B 0,C 180,E1 28565.111,E2 28565.111} C_VEL
LIN {X 0,Y 629.281,Z 1098.757,A -85,B 0,C 180,E1 28562.969,E2 28562.969} C_VEL
LIN {X 0,Y 627.739,Z 1116.375,A -85,B 0,C 180,E1 28560.643,E2 28560.643} C_VEL
LIN {X 0,Y 626.511,Z 1132.303,A -85,B 0,C 180,E1 28558.239,E2 28558.239} C_VEL
LIN {X 0,Y 625.553,Z 1146.48,A -85,B 0,C 180,E1 28555.77,E2 28555.77} C_VEL
LIN {X 0,Y 624.865,Z 1159.213,A -85,B 0,C 180,E1 28553.18,E2 28553.18} C_VEL
LIN {X 0,Y 624.406,Z 1169.316,A -85,B 0,C 180,E1 28550.725,E2 28550.725} C_VEL
LIN {X 0,Y 624.162,Z 1177.029,A -85,B 0,C 180,E1 28548.491,E2 28548.491} C_VEL
LIN {X 0,Y 624.013,Z 1183.792,A -85,B 0,C 180,E1 28546.093,E2 28546.093} C_VEL
LIN {X 0,Y 623.94,Z 1189.017,A -85,B 0,C 180,E1 28543.625,E2 28543.625} C_VEL
LIN {X 0,Y 623.916,Z 1192.349,A -85,B 0,C 180,E1 28541.368,E2 28541.368} C_VEL
LIN {X 0,Y 623.913,Z 1194.398,A -85,B 0,C 180,E1 28539.036,E2 28539.036} C_VEL
LIN {X 0,Y 623.907,Z 1194.883,A -85,B 0,C 180,E1 28536.441,E2 28536.441} C_VEL
LIN {X 0,Y 623.911,Z 1193.959,A -85,B 0,C 180,E1 28534.228,E2 28534.228} C_VEL
LIN {X 0,Y 623.924,Z 1191.601,A -85,B 0,C 180,E1 28531.929,E2 28531.929} C_VEL
LIN {X 0,Y 623.955,Z 1187.427,A -85,B 0,C 180,E1 28529.449,E2 28529.449} C_VEL
LIN {X 0,Y 624.043,Z 1182.044,A -85,B 0,C 180,E1 28527.153,E2 28527.153} C_VEL
LIN {X 0,Y 624.219,Z 1174.963,A -85,B 0,C 180,E1 28524.762,E2 28524.762} C_VEL
LIN {X 0,Y 624.569,Z 1165.395,A -85,B 0,C 180,E1 28522.179,E2 28522.179} C_VEL
LIN {X 0,Y 625.047,Z 1155.178,A -85,B 0,C 180,E1 28519.865,E2 28519.865} C_VEL
LIN {X 0,Y 625.785,Z 1142.716,A -85,B 0,C 180,E1 28517.45,E2 28517.45} C_VEL
LIN {X 0,Y 626.742,Z 1128.8,A -85,B 0,C 180,E1 28515.117,E2 28515.117} C_VEL
LIN {X 0,Y 627.981,Z 1113.514,A -85,B 0,C 180,E1 28512.869,E2 28512.869} C_VEL
LIN {X 0,Y 629.417,Z 1096.824,A -85,B 0,C 180,E1 28510.706,E2 28510.706} C_VEL
LIN {X 0,Y 631.271,Z 1077.903,A -85,B 0,C 180,E1 28508.539,E2 28508.539} C_VEL
LIN {X 0,Y 633.277,Z 1057.74,A -85,B 0,C 180,E1 28506.505,E2 28506.505} C_VEL
LIN {X 0,Y 635.528,Z 1036.529,A -85,B 0,C 180,E1 28504.614,E2 28504.614} C_VEL
LIN {X 0,Y 637.922,Z 1013.499,A -85,B 0,C 180,E1 28502.814,E2 28502.814} C_VEL
LIN {X 0,Y 640.354,Z 989.999,A -85,B 0,C 180,E1 28501.204,E2 28501.204} C_VEL
LIN {X 0,Y 642.844,Z 965.302,A -85,B 0,C 180,E1 28499.739,E2 28499.739} C_VEL
LIN {X 0,Y 644.907,Z 943.235,A -85,B 0,C 180,E1 28498.605,E2 28498.605} C_VEL
LIN {X 0,Y 646.947,Z 920.041,A -85,B 0,C 180,E1 28497.569,E2 28497.569} C_VEL
LIN {X 0,Y 648.961,Z 893.626,A -85,B 0,C 180,E1 28496.578,E2 28496.578} C_VEL
LIN {X 0,Y 650.512,Z 870.496,A -85,B 0,C 180,E1 28495.867,E2 28495.867} C_VEL
LIN {X 0,Y 651.831,Z 847.478,A -85,B 0,C 180,E1 28495.29,E2 28495.29} C_VEL
LIN {X 0,Y 653.079,Z 819.584,A -85,B 0,C 180,E1 28494.761,E2 28494.761} C_VEL
LIN {X 0,Y 656.099,Z 664.899,A -85,B 0,C 180,E1 28492.694,E2 28492.694} C_VEL
LIN {X 0,Y 660.35,Z 449.648,A -85,B 0,C 180,E1 28489.778,E2 28489.778} C_VEL
LIN {X 0,Y 661.426,Z 389.872,A -85,B 0,C 180,E1 28488.936,E2 28488.936} C_VEL
LIN {X 0,Y 650.088,Z 373.083,A -85,B 0,C 180,E1 28487.531,E2 28487.531} C_VEL
LIN {X 0,Y 640.085,Z 359.085,A -85,B 0,C 180,E1 28486.228,E2 28486.228} C_VEL
LIN {X 0,Y 630.01,Z 345.596,A -85,B 0,C 180,E1 28484.868,E2 28484.868} C_VEL
LIN {X 0,Y 627.078,Z 341.251,A -85,B 0,C 180,E1 28484.427,E2 28484.427} C_VEL
LIN {X 0,Y 625.145,Z 337.483,A -85,B 0,C 180,E1 28483.834,E2 28483.834} C_VEL
LIN {X 0,Y 624.933,Z 336.385,A -85,B 0,C 180,E1 28483.683,E2 28483.683} C_VEL
LIN {X 0,Y 624.854,Z 336.392,A -85,B 0,C 180,E1 28480.759,E2 28480.759} C_VEL
LIN {X 0,Y 624.886,Z 336.396,A -85,B 0,C 180,E1 28478.028,E2 28478.028} C_VEL
LIN {X 0,Y 624.865,Z 336.386,A -85,B 0,C 180,E1 28474.829,E2 28474.829} C_VEL
LIN {X 0,Y 624.864,Z 336.388,A -85,B 0,C 180,E1 28472.171,E2 28472.171} C_VEL
LIN {X 0,Y 624.91,Z 336.365,A -85,B 0,C 180,E1 28469.106,E2 28469.106} C_VEL
LIN {X 0,Y 624.858,Z 336.381,A -85,B 0,C 180,E1 28466.312,E2 28466.312} C_VEL
LIN {X 0,Y 624.924,Z 336.369,A -85,B 0,C 180,E1 28463.379,E2 28463.379} C_VEL
LIN {X 0,Y 624.86,Z 336.372,A -85,B 0,C 180,E1 28460.319,E2 28460.319} C_VEL
LIN {X 0,Y 624.881,Z 336.393,A -85,B 0,C 180,E1 28457.603,E2 28457.603} C_VEL
LIN {X 0,Y 624.875,Z 336.388,A -85,B 0,C 180,E1 28454.361,E2 28454.361} C_VEL
LIN {X 0,Y 624.865,Z 336.391,A -85,B 0,C 180,E1 28451.687,E2 28451.687} C_VEL
LIN {X 0,Y 624.918,Z 336.39,A -85,B 0,C 180,E1 28448.558,E2 28448.558} C_VEL
LIN {X 0,Y 624.862,Z 336.383,A -85,B 0,C 180,E1 28445.786,E2 28445.786} C_VEL
LIN {X 0,Y 624.915,Z 336.382,A -85,B 0,C 180,E1 28442.935,E2 28442.935} C_VEL
LIN {X 0,Y 624.873,Z 336.386,A -85,B 0,C 180,E1 28439.908,E2 28439.908} C_VEL
LIN {X 0,Y 624.872,Z 336.391,A -85,B 0,C 180,E1 28437.248,E2 28437.248} C_VEL
LIN {X 0,Y 624.913,Z 336.39,A -85,B 0,C 180,E1 28434.122,E2 28434.122} C_VEL
LIN {X 0,Y 624.866,Z 336.386,A -85,B 0,C 180,E1 28431.349,E2 28431.349} C_VEL
LIN {X 0,Y 624.941,Z 336.356,A -85,B 0,C 180,E1 28428.37,E2 28428.37} C_VEL
LIN {X 0,Y 624.869,Z 336.383,A -85,B 0,C 180,E1 28425.355,E2 28425.355} C_VEL
LIN {X 0,Y 624.897,Z 336.376,A -85,B 0,C 180,E1 28422.589,E2 28422.589} C_VEL
LIN {X 0,Y 624.88,Z 336.375,A -85,B 0,C 180,E1 28419.388,E2 28419.388} C_VEL
LIN {X 0,Y 624.871,Z 336.383,A -85,B 0,C 180,E1 28416.819,E2 28416.819} C_VEL
LIN {X 0,Y 624.943,Z 336.363,A -85,B 0,C 180,E1 28413.794,E2 28413.794} C_VEL
LIN {X 0,Y 624.873,Z 336.389,A -85,B 0,C 180,E1 28410.886,E2 28410.886} C_VEL
LIN {X 0,Y 624.91,Z 336.388,A -85,B 0,C 180,E1 28408.128,E2 28408.128} C_VEL
LIN {X 0,Y 624.883,Z 336.394,A -85,B 0,C 180,E1 28404.939,E2 28404.939} C_VEL
LIN {X 0,Y 624.924,Z 336.493,A -85,B 0,C 180,E1 28404.02,E2 28404.02} C_VEL
LIN {X 0,Y 626.19,Z 339.772,A -85,B 0,C 180,E1 28403.558,E2 28403.558} C_VEL
LIN {X 0,Y 627.188,Z 341.436,A -85,B 0,C 180,E1 28403.284,E2 28403.284} C_VEL
LIN {X 0,Y 631.833,Z 350.576,A -85,B 0,C 180,E1 28401.947,E2 28401.947} C_VEL
LIN {X 0,Y 646.023,Z 370.391,A -85,B 0,C 180,E1 28400.049,E2 28400.049} C_VEL
LIN {X 0,Y 658.686,Z 388.838,A -85,B 0,C 180,E1 28398.457,E2 28398.457} C_VEL
LIN {X 0,Y 661.686,Z 393.531,A -85,B 0,C 180,E1 28398.091,E2 28398.091} C_VEL
